C07274=1119.988,-13.062,-50.187,179.666,6.143,149.206
C07275=1119.993,-13.312,-50.175,179.666,6.138,149.205
C07276=1119.998,-13.562,-50.161,179.665,6.134,149.204
C07277=1120.003,-13.811,-50.149,179.664,6.129,149.203
C07278=1120.008,-14.061,-50.136,179.664,6.125,149.202
C07279=1120.013,-14.311,-50.123,179.663,6.120,149.202
C07280=1120.019,-14.560,-50.110,179.663,6.115,149.201
C07281=1120.023,-14.809,-50.096,179.662,6.111,149.200
C07282=1120.029,-15.058,-50.084,179.661,6.106,149.199
C07283=1120.034,-15.309,-50.070,179.661,6.101,149.198
C07284=1120.039,-15.558,-50.058,179.660,6.097,149.197
C07285=1120.044,-15.808,-50.046,179.659,6.092,149.197
C07286=1120.049,-16.058,-50.033,179.659,6.088,149.196
C07287=1120.055,-16.308,-50.020,179.658,6.082,149.195
C07288=1120.060,-16.557,-50.007,179.657,6.077,149.194
C07289=1120.065,-16.806,-49.994,179.656,6.073,149.193
C07290=1120.070,-17.056,-49.981,179.656,6.068,149.192
C07291=1120.075,-17.306,-49.968,179.655,6.064,149.192
C07292=1120.081,-17.555,-49.956,179.655,6.059,149.191
C07293=1120.085,-17.805,-49.943,179.654,6.054,149.190
C07294=1120.090,-18.054,-49.930,179.653,6.050,149.189
C07295=1120.095,-18.304,-49.918,179.653,6.045,149.188
C07296=1120.101,-18.553,-49.904,179.652,6.040,149.187
C07297=1120.106,-18.803,-49.891,179.652,6.036,149.186
C07298=1120.111,-19.053,-49.879,179.651,6.031,149.186
C07299=1120.116,-19.268,-49.868,179.650,6.026,149.185
C07300=1120.120,-19.484,-49.858,179.650,6.023,149.184
C07301=1120.124,-19.698,-49.846,179.649,6.019,149.183
C07302=1120.130,-19.913,-49.836,179.649,6.015,149.183
C07303=1120.133,-20.128,-49.825,179.648,6.010,149.182
C07304=1120.138,-20.343,-49.814,179.647,6.006,149.181
C07305=1120.143,-20.558,-49.803,179.647,6.002,149.181
C07306=1120.147,-20.774,-49.792,179.646,5.998,149.180
C07307=1120.152,-21.023,-49.780,179.645,5.993,149.179
C07308=1120.158,-21.272,-49.767,179.645,5.989,149.178
C07309=1120.163,-21.522,-49.755,179.644,5.984,149.177
C07310=1120.167,-21.772,-49.742,179.644,5.979,149.176
C07311=1120.173,-22.022,-49.729,179.643,5.974,149.175
C07312=1120.178,-22.271,-49.717,179.643,5.970,149.175
C07313=1120.183,-22.521,-49.705,179.642,5.964,149.174
C07314=1120.188,-22.770,-49.692,179.641,5.960,149.173
C07315=1120.193,-23.020,-49.680,179.640,5.955,149.172
C07316=1120.199,-23.270,-49.668,179.640,5.950,149.171
C07317=1120.203,-23.520,-49.655,179.640,5.946,149.170
C07318=1120.208,-23.769,-49.642,179.638,5.940,149.169
C07319=1120.215,-24.019,-49.630,179.638,5.935,149.168
C07320=1120.220,-24.268,-49.617,179.637,5.931,149.168
C07321=1120.225,-24.518,-49.604,179.637,5.926,149.167
C07322=1120.230,-24.768,-49.593,179.637,5.921,149.166
C07323=1120.235,-25.017,-49.580,179.635,5.916,149.165
C07324=1120.241,-25.266,-49.567,179.635,5.911,149.164
C07325=1120.245,-25.517,-49.555,179.635,5.906,149.163
C07326=1120.251,-25.766,-49.542,179.634,5.902,149.162
C07327=1120.256,-26.016,-49.531,179.634,5.897,149.161
C07328=1120.261,-26.266,-49.518,179.634,5.892,149.160
C07329=1120.266,-26.515,-49.507,179.635,5.889,149.159
C07330=1120.271,-26.764,-49.494,179.636,5.884,149.158
C07331=1120.276,-27.014,-49.481,179.636,5.880,149.157
C07332=1120.281,-27.264,-49.470,179.637,5.876,149.156
C07333=1120.287,-27.513,-49.457,179.637,5.872,149.155
C07334=1120.292,-27.763,-49.445,179.638,5.868,149.154
C07335=1120.297,-28.013,-49.432,179.638,5.864,149.153
C07336=1120.302,-28.263,-49.420,179.639,5.859,149.152
C07337=1120.307,-28.512,-49.408,179.639,5.855,149.151
C07338=1120.313,-28.762,-49.396,179.640,5.851,149.150
C07339=1120.318,-29.012,-49.383,179.640,5.847,149.149
C07340=1120.323,-29.261,-49.371,179.640,5.843,149.148
C07341=1120.328,-29.511,-49.359,179.640,5.839,149.147
C07342=1120.334,-29.761,-49.347,179.641,5.835,149.146
C07343=1120.339,-30.010,-49.334,179.641,5.831,149.145
C07344=1120.344,-30.260,-49.322,179.641,5.826,149.144
C07345=1120.349,-30.509,-49.310,179.641,5.822,149.143
C07346=1120.354,-30.759,-49.298,179.641,5.818,149.142
C07347=1120.359,-31.008,-49.286,179.641,5.813,149.141
C07348=1120.365,-31.258,-49.274,179.641,5.809,149.140
C07349=1120.370,-31.507,-49.261,179.641,5.805,149.139
C07350=1120.375,-31.757,-49.249,179.641,5.800,149.138
C07351=1120.381,-32.007,-49.238,179.641,5.796,149.137
C07352=1120.386,-32.257,-49.225,179.641,5.791,149.136
C07353=1120.390,-32.506,-49.214,179.641,5.787,149.135
C07354=1120.395,-32.756,-49.201,179.640,5.783,149.135
C07355=1120.400,-32.972,-49.190,179.640,5.779,149.134
C07356=1120.404,-33.186,-49.180,179.640,5.776,149.133
C07357=1120.409,-33.402,-49.170,179.640,5.772,149.132
C07358=1120.414,-33.616,-49.160,179.639,5.767,149.131
C07359=1120.417,-33.832,-49.149,179.638,5.764,149.131
C07360=1120.422,-34.047,-49.139,179.638,5.760,149.130
C07361=1120.427,-34.262,-49.129,179.638,5.756,149.129
C07362=1120.432,-34.477,-49.118,179.637,5.752,149.129
C07363=1120.437,-34.727,-49.107,179.637,5.747,149.128
C07364=1120.442,-34.976,-49.094,179.636,5.743,149.127
C07365=1120.447,-35.226,-49.082,179.635,5.738,149.126
C07366=1120.453,-35.476,-49.070,179.635,5.733,149.125
C07367=1120.458,-35.725,-49.058,179.634,5.729,149.124
C07368=1120.462,-35.975,-49.046,179.634,5.724,149.124
C07369=1120.468,-36.225,-49.034,179.633,5.719,149.123
C07370=1120.473,-36.474,-49.022,179.632,5.715,149.122
C07371=1120.478,-36.724,-49.010,179.632,5.710,149.121
C07372=1120.483,-36.974,-48.999,179.631,5.705,149.120
C07373=1120.489,-37.224,-48.987,179.630,5.700,149.120
C07374=1120.494,-37.474,-48.975,179.629,5.696,149.119
C07375=1120.499,-37.723,-48.962,179.628,5.691,149.118
C07376=1120.504,-37.973,-48.951,179.627,5.686,149.117
C07377=1120.509,-38.223,-48.939,179.626,5.681,149.116
C07378=1120.515,-38.472,-48.928,179.625,5.676,149.115
C07379=1120.520,-38.721,-48.916,179.624,5.671,149.115
C07380=1120.525,-38.971,-48.904,179.623,5.666,149.114
C07381=1120.530,-39.221,-48.892,179.622,5.661,149.113
C07382=1120.535,-39.470,-48.881,179.621,5.655,149.112
C07383=1120.541,-39.720,-48.869,179.620,5.651,149.112
C07384=1120.546,-39.970,-48.857,179.619,5.645,149.111
C07385=1120.551,-40.220,-48.846,179.617,5.640,149.110
C07386=1120.557,-40.469,-48.834,179.616,5.635,149.109
C07387=1120.562,-40.719,-48.822,179.615,5.630,149.109
C07388=1120.567,-40.969,-48.811,179.614,5.624,149.108
C07389=1120.572,-41.219,-48.799,179.612,5.619,149.107
C07390=1120.578,-41.468,-48.787,179.611,5.613,149.106
C07391=1120.582,-41.718,-48.776,179.610,5.608,149.105
C07392=1120.588,-41.967,-48.764,179.609,5.603,149.104
C07393=1120.593,-42.217,-48.753,179.607,5.597,149.104
C07394=1120.599,-42.467,-48.741,179.605,5.591,149.103
C07395=1120.603,-42.717,-48.730,179.604,5.586,149.102
C07396=1120.609,-42.966,-48.718,179.603,5.580,149.101
C07397=1120.614,-43.215,-48.707,179.602,5.576,149.100
C07398=1120.619,-43.465,-48.695,179.602,5.570,149.099
C07399=1120.624,-43.715,-48.684,179.603,5.565,149.098
C07400=1120.630,-43.965,-48.672,179.603,5.561,149.097
C07401=1120.635,-44.215,-48.660,179.603,5.556,149.096
C07402=1120.640,-44.464,-48.649,179.603,5.552,149.095
C07403=1120.646,-44.714,-48.637,179.603,5.547,149.094
C07404=1120.650,-44.963,-48.626,179.603,5.542,149.093
C07405=1120.655,-45.214,-48.615,179.604,5.538,149.092
C07406=1120.661,-45.463,-48.604,179.604,5.533,149.091
C07407=1120.666,-45.712,-48.593,179.604,5.528,149.089
C07408=1120.672,-45.962,-48.581,179.604,5.523,149.089
C07409=1120.676,-46.212,-48.569,179.604,5.518,149.087
C07410=1120.682,-46.461,-48.558,179.605,5.514,149.086
C07411=1120.687,-46.677,-48.549,179.605,5.510,149.085
C07412=1120.691,-46.892,-48.538,179.605,5.506,149.084
C07413=1120.695,-47.108,-48.529,179.605,5.501,149.084
C07414=1120.700,-47.323,-48.519,179.605,5.497,149.083
C07415=1120.704,-47.538,-48.510,179.605,5.493,149.082
C07416=1120.709,-47.753,-48.500,179.605,5.490,149.081
C07417=1120.714,-47.968,-48.489,179.605,5.486,149.080
C07418=1120.718,-48.184,-48.480,179.606,5.482,149.079
C07419=1120.723,-48.433,-48.468,179.606,5.476,149.078
C07420=1120.728,-48.682,-48.458,179.606,5.472,149.077
C07421=1120.734,-48.933,-48.446,179.606,5.467,149.076
C07422=1120.739,-49.182,-48.435,179.607,5.463,149.075
C07423=1120.745,-49.432,-48.424,179.607,5.458,149.073
C07424=1120.749,-49.681,-48.412,179.607,5.453,149.072
C07425=1120.754,-49.931,-48.402,179.607,5.449,149.071
C07426=1120.760,-50.181,-48.390,179.607,5.444,149.070
C07427=1120.765,-50.430,-48.379,179.608,5.439,149.069
C07428=1120.771,-50.680,-48.367,179.607,5.435,149.068
C07429=1120.776,-50.930,-48.357,179.608,5.430,149.067
C07430=1120.781,-51.179,-48.345,179.608,5.425,149.066
C07431=1120.786,-51.429,-48.334,179.608,5.420,149.065
C07432=1120.792,-51.679,-48.323,179.608,5.416,149.064
C07433=1120.797,-51.929,-48.312,179.608,5.411,149.063
C07434=1120.802,-52.178,-48.300,179.609,5.407,149.062
C07435=1120.808,-52.428,-48.290,179.609,5.402,149.061
C07436=1120.812,-52.678,-48.279,179.609,5.397,149.060
C07437=1120.818,-52.928,-48.267,179.609,5.392,149.058
C07438=1120.823,-53.177,-48.257,179.609,5.388,149.057
C07439=1120.828,-53.427,-48.245,179.610,5.383,149.056
C07440=1120.834,-53.677,-48.234,179.610,5.378,149.055
C07441=1120.839,-53.926,-48.223,179.609,5.373,149.054
C07442=1120.844,-54.176,-48.212,179.610,5.369,149.053
C07443=1120.849,-54.426,-48.201,179.610,5.364,149.052
C07444=1120.855,-54.675,-48.190,179.610,5.360,149.051
C07445=1120.859,-54.925,-48.179,179.610,5.355,149.050
C07446=1120.865,-55.175,-48.168,179.611,5.350,149.049
C07447=1120.871,-55.424,-48.156,179.611,5.346,149.048
C07448=1120.876,-55.675,-48.146,179.611,5.341,149.047
C07449=1120.881,-55.924,-48.135,179.611,5.336,149.045
C07450=1120.886,-56.174,-48.124,179.611,5.331,149.045
C07451=1120.891,-56.424,-48.112,179.612,5.327,149.043
C07452=1120.897,-56.673,-48.102,179.612,5.322,149.042
C07453=1120.902,-56.923,-48.091,179.612,5.318,149.041
C07454=1120.907,-57.173,-48.081,179.612,5.313,149.040
C07455=1120.912,-57.422,-48.069,179.612,5.308,149.039
C07456=1120.917,-57.672,-48.058,179.612,5.304,149.038
C07457=1120.923,-57.922,-48.047,179.612,5.299,149.037
C07458=1120.928,-58.172,-48.037,179.613,5.295,149.036
C07459=1120.933,-58.421,-48.026,179.613,5.289,149.035
C07460=1120.938,-58.671,-48.015,179.613,5.284,149.034
C07461=1120.944,-58.920,-48.004,179.613,5.280,149.033
C07462=1120.949,-59.171,-47.993,179.613,5.275,149.032
C07463=1120.954,-59.420,-47.982,179.614,5.271,149.031
C07464=1120.959,-59.670,-47.972,179.613,5.266,149.030
C07465=1120.964,-59.919,-47.960,179.614,5.262,149.028
C07466=1120.970,-60.169,-47.950,179.614,5.257,149.028
C07467=1120.974,-60.384,-47.941,179.613,5.252,149.027
C07468=1120.979,-60.600,-47.932,179.612,5.248,149.026
C07469=1120.983,-60.815,-47.922,179.612,5.243,149.025
C07470=1120.988,-61.030,-47.912,179.611,5.239,149.024
C07471=1120.993,-61.246,-47.903,179.610,5.234,149.024
C07472=1120.997,-61.461,-47.894,179.610,5.230,149.023
C07473=1121.001,-61.676,-47.885,179.609,5.225,149.022
C07474=1121.006,-61.892,-47.876,179.609,5.221,149.021
C07475=1121.011,-62.141,-47.865,179.608,5.216,149.020
C07476=1121.016,-62.391,-47.854,179.607,5.210,149.019
C07477=1121.022,-62.641,-47.844,179.607,5.205,149.018
C07478=1121.027,-62.890,-47.832,179.606,5.200,149.017
C07479=1121.033,-63.140,-47.822,179.606,5.195,149.017
C07480=1121.038,-63.390,-47.811,179.605,5.190,149.016
C07481=1121.043,-63.640,-47.801,179.605,5.184,149.014
C07482=1121.048,-63.889,-47.790,179.604,5.179,149.014
C07483=1121.054,-64.139,-47.780,179.603,5.174,149.013
C07484=1121.059,-64.389,-47.770,179.602,5.169,149.012
C07485=1121.064,-64.639,-47.759,179.602,5.164,149.011
C07486=1121.070,-64.888,-47.748,179.601,5.158,149.010
C07487=1121.075,-65.138,-47.737,179.601,5.153,149.009
C07488=1121.080,-65.387,-47.727,179.600,5.147,149.008
C07489=1121.085,-65.638,-47.717,179.600,5.142,149.007
C07490=1121.090,-65.887,-47.706,179.599,5.137,149.006
C07491=1121.096,-66.136,-47.696,179.599,5.132,149.005
C07492=1121.101,-66.386,-47.685,179.598,5.126,149.004
C07493=1121.107,-66.636,-47.675,179.598,5.121,149.003
C07494=1121.112,-66.886,-47.664,179.598,5.117,149.002
C07495=1121.117,-67.136,-47.654,179.597,5.111,149.001
C07496=1121.123,-67.385,-47.644,179.597,5.106,149.000
C07497=1121.128,-67.635,-47.632,179.596,5.100,148.999
C07498=1121.133,-67.884,-47.622,179.596,5.095,148.998
C07499=1121.138,-68.135,-47.612,179.596,5.089,148.997
C07500=1121.143,-68.384,-47.602,179.595,5.084,148.996
C07501=1121.149,-68.634,-47.592,179.595,5.080,148.995
C07502=1121.154,-68.884,-47.581,179.594,5.074,148.994
C07503=1121.159,-69.133,-47.571,179.594,5.069,148.992
C07504=1121.165,-69.383,-47.561,179.594,5.064,148.991
C07505=1121.170,-69.633,-47.550,179.594,5.058,148.990
C07506=1121.175,-69.883,-47.540,179.593,5.053,148.989
C07507=1121.181,-70.132,-47.530,179.593,5.047,148.988
C07508=1121.186,-70.382,-47.519,179.592,5.042,148.987
C07509=1121.191,-70.632,-47.510,179.593,5.037,148.986
C07510=1121.196,-70.881,-47.499,179.592,5.031,148.985
C07511=1121.201,-71.131,-47.489,179.592,5.026,148.984
C07512=1121.207,-71.381,-47.479,179.592,5.021,148.983
C07513=1121.213,-71.631,-47.468,179.591,5.017,148.982
C07514=1121.218,-71.881,-47.458,179.591,5.011,148.981
C07515=1121.223,-72.130,-47.448,179.591,5.005,148.980
C07516=1121.228,-72.380,-47.438,179.591,5.000,148.978
C07517=1121.233,-72.630,-47.428,179.590,4.995,148.978
C07518=1121.239,-72.879,-47.417,179.590,4.990,148.976
C07519=1121.245,-73.130,-47.408,179.591,4.984,148.975
C07520=1121.250,-73.379,-47.398,179.590,4.980,148.974
C07521=1121.254,-73.629,-47.388,179.590,4.974,148.973
C07522=1121.260,-73.879,-47.377,179.590,4.968,148.972
C07523=1121.265,-74.094,-47.368,179.590,4.965,148.971
C07524=1121.269,-74.309,-47.361,179.590,4.960,148.970
C07525=1121.274,-74.525,-47.351,179.589,4.955,148.969
C07526=1121.278,-74.740,-47.343,179.590,4.951,148.968
C07527=1121.283,-74.956,-47.334,179.590,4.946,148.967
C07528=1121.287,-75.170,-47.326,179.590,4.942,148.966
C07529=1121.292,-75.386,-47.317,179.590,4.937,148.965
C07530=1121.297,-75.602,-47.308,179.589,4.932,148.964
C07531=1121.302,-75.851,-47.298,179.590,4.927,148.963
C07532=1121.308,-76.101,-47.288,179.590,4.922,148.962
C07533=1121.313,-76.351,-47.278,179.590,4.917,148.961
C07534=1121.318,-76.601,-47.268,179.590,4.912,148.960
C07535=1121.323,-76.850,-47.258,179.590,4.907,148.958
C07536=1121.329,-77.100,-47.248,179.590,4.902,148.958
C07537=1121.335,-77.350,-47.239,179.589,4.896,148.956
C07538=1121.340,-77.599,-47.229,179.590,4.891,148.955
C07539=1121.345,-77.850,-47.218,179.590,4.886,148.954
C07540=1121.350,-78.099,-47.208,179.590,4.880,148.953
C07541=1121.355,-78.349,-47.199,179.590,4.875,148.952
C07542=1121.361,-78.599,-47.189,179.590,4.870,148.951
C07543=1121.367,-78.848,-47.179,179.590,4.865,148.949
C07544=1121.372,-79.098,-47.170,179.590,4.860,148.948
C07545=1121.377,-79.348,-47.159,179.591,4.855,148.947
C07546=1121.382,-79.597,-47.150,179.591,4.849,148.946
C07547=1121.388,-79.848,-47.140,179.591,4.844,148.945
C07548=1121.393,-80.097,-47.130,179.591,4.839,148.944
C07549=1121.398,-80.346,-47.120,179.591,4.834,148.942
C07550=1121.404,-80.596,-47.111,179.591,4.829,148.941
C07551=1121.410,-80.846,-47.101,179.592,4.824,148.940
C07552=1121.414,-81.097,-47.091,179.592,4.819,148.939
C07553=1121.420,-81.346,-47.081,179.592,4.813,148.938
C07554=1121.425,-81.595,-47.072,179.592,4.808,148.936
C07555=1121.430,-81.846,-47.062,179.592,4.803,148.935
C07556=1121.435,-82.095,-47.053,179.592,4.798,148.934
C07557=1121.441,-82.345,-47.043,179.593,4.793,148.933
C07558=1121.447,-82.594,-47.033,179.593,4.788,148.932
C07559=1121.451,-82.844,-47.023,179.594,4.783,148.930
C07560=1121.457,-83.095,-47.013,179.594,4.778,148.929
C07561=1121.462,-83.344,-47.004,179.594,4.773,148.928
C07562=1121.468,-83.594,-46.994,179.595,4.767,148.927
C07563=1121.473,-83.843,-46.985,179.595,4.762,148.926
C07564=1121.479,-84.093,-46.975,179.595,4.757,148.925
C07565=1121.483,-84.343,-46.966,179.596,4.753,148.923
C07566=1121.489,-84.593,-46.956,179.596,4.748,148.922
C07567=1121.494,-84.842,-46.946,179.596,4.742,148.921
C07568=1121.500,-85.092,-46.937,179.597,4.737,148.920
C07569=1121.505,-85.341,-46.927,179.597,4.732,148.918
C07570=1121.510,-85.592,-46.917,179.598,4.727,148.917
C07571=1121.515,-85.841,-46.908,179.598,4.722,148.916
C07572=1121.521,-86.092,-46.898,179.598,4.717,148.915
C07573=1121.526,-86.341,-46.889,179.598,4.712,148.914
C07574=1121.532,-86.591,-46.879,179.599,4.707,148.912
C07575=1121.537,-86.840,-46.870,179.600,4.702,148.911
C07576=1121.543,-87.090,-46.860,179.600,4.697,148.910
C07577=1121.548,-87.340,-46.851,179.601,4.692,148.909
C07578=1121.553,-87.589,-46.842,179.601,4.687,148.908
C07579=1121.557,-87.806,-46.833,179.602,4.683,148.906
C07580=1121.562,-88.021,-46.825,179.602,4.679,148.905
C07581=1121.567,-88.236,-46.817,179.603,4.675,148.904
C07582=1121.572,-88.451,-46.809,179.602,4.670,148.903
C07583=1121.576,-88.667,-46.801,179.603,4.665,148.902
C07584=1121.580,-88.883,-46.793,179.603,4.662,148.901
C07585=1121.585,-89.098,-46.785,179.604,4.657,148.900
C07586=1121.590,-89.314,-46.776,179.604,4.653,148.899
C07587=1121.595,-89.563,-46.767,179.605,4.648,148.898
C07588=1121.601,-89.813,-46.757,179.605,4.644,148.897
C07589=1121.606,-90.063,-46.748,179.606,4.638,148.895
C07590=1121.611,-90.313,-46.739,179.607,4.634,148.894
C07591=1121.617,-90.563,-46.729,179.607,4.629,148.893
C07592=1121.622,-90.813,-46.720,179.608,4.624,148.892
C07593=1121.627,-91.062,-46.711,179.608,4.619,148.890
C07594=1121.633,-91.312,-46.701,179.609,4.614,148.889
C07595=1121.638,-91.562,-46.692,179.609,4.609,148.888
C07596=1121.643,-91.811,-46.682,179.610,4.605,148.887
C07597=1121.649,-92.061,-46.673,179.610,4.600,148.886
C07598=1121.654,-92.311,-46.664,179.612,4.595,148.884
C07599=1121.659,-92.561,-46.654,179.612,4.590,148.883
C07600=1121.664,-92.810,-46.645,179.613,4.585,148.882
C07601=1121.670,-93.060,-46.636,179.613,4.581,148.881
C07602=1121.676,-93.310,-46.627,179.614,4.576,148.879
C07603=1121.680,-93.560,-46.617,179.615,4.571,148.878
C07604=1121.686,-93.810,-46.608,179.615,4.566,148.877
C07605=1121.691,-94.060,-46.599,179.616,4.562,148.876
C07606=1121.697,-94.310,-46.590,179.617,4.557,148.874
C07607=1121.701,-94.559,-46.580,179.617,4.552,148.873
C07608=1121.708,-94.808,-46.571,179.618,4.548,148.872
C07609=1121.713,-95.058,-46.562,179.618,4.543,148.871
C07610=1121.718,-95.308,-46.553,179.618,4.537,148.870
C07611=1121.723,-95.557,-46.544,179.618,4.532,148.869
C07612=1121.729,-95.807,-46.534,179.619,4.528,148.867
C07613=1121.734,-96.057,-46.525,179.619,4.523,148.866
C07614=1121.739,-96.307,-46.517,179.620,4.518,148.865
C07615=1121.745,-96.557,-46.507,179.620,4.512,148.864
C07616=1121.750,-96.807,-46.498,179.620,4.507,148.863
C07617=1121.755,-97.056,-46.489,179.621,4.503,148.861
C07618=1121.761,-97.306,-46.480,179.621,4.498,148.860
C07619=1121.766,-97.556,-46.470,179.621,4.493,148.859
C07620=1121.772,-97.806,-46.461,179.621,4.487,148.858
C07621=1121.777,-98.055,-46.453,179.622,4.483,148.857
C07622=1121.783,-98.305,-46.444,179.622,4.478,148.856
C07623=1121.788,-98.555,-46.434,179.622,4.473,148.855
C07624=1121.794,-98.805,-46.425,179.622,4.468,148.853
C07625=1121.798,-99.054,-46.416,179.623,4.463,148.852
C07626=1121.804,-99.304,-46.407,179.623,4.458,148.851
C07627=1121.810,-99.554,-46.397,179.624,4.453,148.850
C07628=1121.815,-99.804,-46.389,179.624,4.448,148.849
C07629=1121.820,-100.053,-46.380,179.624,4.443,148.847
C07630=1121.826,-100.303,-46.371,179.624,4.438,148.846
C07631=1121.831,-100.553,-46.362,179.625,4.433,148.845
C07632=1121.837,-100.803,-46.353,179.625,4.428,148.844
C07633=1121.842,-101.053,-46.344,179.625,4.423,148.843
C07634=1121.847,-101.303,-46.335,179.625,4.418,148.842
C07635=1121.852,-101.518,-46.327,179.626,4.414,148.840
C07636=1121.856,-101.734,-46.319,179.626,4.409,148.840
C07637=1121.861,-101.949,-46.312,179.626,4.405,148.839
C07638=1121.865,-102.165,-46.304,179.626,4.401,148.838
C07639=1121.870,-102.381,-46.297,179.627,4.396,148.836
C07640=1121.874,-102.596,-46.289,179.627,4.392,148.835
C07641=1121.879,-102.811,-46.281,179.627,4.388,148.835
C07642=1121.883,-103.027,-46.273,179.627,4.383,148.834
C07643=1121.889,-103.276,-46.265,179.627,4.378,148.832
C07644=1121.895,-103.527,-46.255,179.628,4.374,148.831
C07645=1121.900,-103.776,-46.246,179.628,4.369,148.830
C07646=1121.906,-104.027,-46.238,179.628,4.363,148.829
C07647=1121.911,-104.277,-46.229,179.629,4.358,148.828
C07648=1121.917,-104.526,-46.221,179.629,4.353,148.826
C07649=1121.922,-104.776,-46.212,179.629,4.348,148.825
C07650=1121.927,-105.026,-46.203,179.629,4.343,148.824
C07651=1121.932,-105.275,-46.194,179.630,4.338,148.823
C07652=1121.937,-105.525,-46.185,179.630,4.332,148.822
C07653=1121.943,-105.774,-46.177,179.630,4.327,148.820
C07654=1121.948,-106.024,-46.168,179.631,4.323,148.819
C07655=1121.953,-106.274,-46.159,179.631,4.318,148.818
C07656=1121.959,-106.525,-46.151,179.631,4.313,148.817
C07657=1121.964,-106.774,-46.142,179.631,4.308,148.816
C07658=1121.971,-107.024,-46.133,179.631,4.303,148.815
C07659=1121.976,-107.274,-46.124,179.632,4.297,148.814
C07660=1121.981,-107.524,-46.115,179.632,4.292,148.812
C07661=1121.986,-107.773,-46.106,179.632,4.287,148.811
C07662=1121.992,-108.023,-46.098,179.632,4.282,148.810
C07663=1121.997,-108.273,-46.089,179.633,4.277,148.809
C07664=1122.002,-108.523,-46.080,179.633,4.272,148.808
C07665=1122.008,-108.773,-46.071,179.633,4.266,148.806
C07666=1122.013,-109.022,-46.063,179.633,4.261,148.805
C07667=1122.019,-109.272,-46.055,179.634,4.256,148.804
C07668=1122.024,-109.522,-46.046,179.634,4.251,148.803
C07669=1122.030,-109.771,-46.037,179.634,4.246,148.802
C07670=1122.034,-110.021,-46.029,179.634,4.241,148.800
C07671=1122.040,-110.271,-46.021,179.635,4.235,148.799
C07672=1122.045,-110.521,-46.012,179.635,4.230,148.798
C07673=1122.051,-110.770,-46.003,179.635,4.225,148.797
C07674=1122.056,-111.020,-45.994,179.635,4.220,148.796
C07675=1122.061,-111.271,-45.986,179.636,4.215,148.794
C07676=1122.067,-111.520,-45.978,179.636,4.210,148.793
C07677=1122.072,-111.770,-45.969,179.636,4.204,148.792
C07678=1122.078,-112.020,-45.961,179.636,4.199,148.791
C07679=1122.083,-112.269,-45.952,179.636,4.194,148.790
C07680=1122.089,-112.519,-45.943,179.636,4.189,148.789
C07681=1122.094,-112.770,-45.935,179.637,4.184,148.787
C07682=1122.100,-113.019,-45.926,179.637,4.179,148.786
C07683=1122.105,-113.269,-45.918,179.637,4.174,148.785
C07684=1122.110,-113.519,-45.910,179.637,4.169,148.784
C07685=1122.116,-113.768,-45.901,179.638,4.163,148.783
C07686=1122.121,-114.018,-45.893,179.638,4.158,148.781
C07687=1122.126,-114.268,-45.884,179.638,4.152,148.780
C07688=1122.132,-114.517,-45.876,179.638,4.147,148.779
C07689=1122.137,-114.768,-45.868,179.638,4.142,148.778
C07690=1122.143,-115.017,-45.859,179.638,4.137,148.777
C07691=1122.147,-115.233,-45.852,179.639,4.132,148.775
C07692=1122.152,-115.448,-45.845,179.639,4.128,148.774
C07693=1122.157,-115.664,-45.838,179.639,4.124,148.773
C07694=1122.161,-115.880,-45.830,179.640,4.118,148.772
C07695=1122.166,-116.096,-45.823,179.639,4.114,148.771
C07696=1122.171,-116.311,-45.816,179.640,4.109,148.770
C07697=1122.175,-116.527,-45.809,179.640,4.104,148.769
C07698=1122.180,-116.742,-45.802,179.640,4.101,148.768
C07699=1122.185,-116.992,-45.793,179.641,4.095,148.767
C07700=1122.191,-117.242,-45.785,179.641,4.090,148.766
C07701=1122.196,-117.492,-45.776,179.641,4.084,148.765
C07702=1122.202,-117.741,-45.769,179.641,4.079,148.763
C07703=1122.207,-117.991,-45.760,179.641,4.074,148.762
C07704=1122.213,-118.241,-45.752,179.641,4.069,148.761
C07705=1122.218,-118.491,-45.744,179.642,4.063,148.759
C07706=1122.223,-118.741,-45.736,179.642,4.058,148.758
C07707=1122.229,-118.991,-45.728,179.642,4.052,148.757
C07708=1122.234,-119.241,-45.719,179.642,4.047,148.756
C07709=1122.240,-119.490,-45.711,179.643,4.042,148.755
C07710=1122.245,-119.740,-45.703,179.643,4.036,148.753
C07711=1122.251,-119.990,-45.695,179.643,4.031,148.752
C07712=1122.256,-120.240,-45.687,179.643,4.025,148.751
C07713=1122.262,-120.489,-45.678,179.643,4.020,148.750
C07714=1122.267,-120.739,-45.671,179.643,4.015,148.749
C07715=1122.272,-120.989,-45.662,179.644,4.010,148.747
C07716=1122.278,-121.239,-45.654,179.643,4.004,148.746
C07717=1122.283,-121.489,-45.647,179.644,3.998,148.745
C07718=1122.288,-121.738,-45.638,179.645,3.993,148.744
C07719=1122.294,-121.989,-45.630,179.645,3.988,148.742
C07720=1122.299,-122.238,-45.623,179.645,3.982,148.741
C07721=1122.304,-122.488,-45.614,179.645,3.977,148.740
C07722=1122.310,-122.738,-45.606,179.645,3.971,148.739
C07723=1122.315,-122.988,-45.598,179.645,3.966,148.737
C07724=1122.321,-123.237,-45.590,179.646,3.960,148.736
C07725=1122.326,-123.488,-45.582,179.646,3.955,148.735
C07726=1122.332,-123.737,-45.574,179.646,3.950,148.734
C07727=1122.338,-123.987,-45.567,179.647,3.944,148.732
C07728=1122.343,-124.237,-45.558,179.646,3.938,148.731
C07729=1122.348,-124.486,-45.551,179.647,3.933,148.730
C07730=1122.354,-124.737,-45.542,179.647,3.928,148.729
C07731=1122.359,-124.986,-45.535,179.647,3.922,148.727
C07732=1122.364,-125.236,-45.526,179.647,3.916,148.726
C07733=1122.370,-125.486,-45.518,179.648,3.911,148.725
C07734=1122.375,-125.736,-45.511,179.647,3.905,148.724
C07735=1122.381,-125.986,-45.503,179.648,3.900,148.722
C07736=1122.386,-126.235,-45.495,179.649,3.895,148.721
C07737=1122.392,-126.485,-45.487,179.648,3.889,148.720
C07738=1122.397,-126.735,-45.480,179.649,3.883,148.719
C07739=1122.402,-126.985,-45.471,179.648,3.877,148.717
C07740=1122.408,-127.234,-45.464,179.649,3.872,148.716
C07741=1122.413,-127.485,-45.456,179.649,3.867,148.715
C07742=1122.419,-127.734,-45.448,179.649,3.861,148.713
C07743=1122.424,-127.984,-45.440,179.649,3.855,148.712
C07744=1122.430,-128.234,-45.432,179.649,3.849,148.711
C07745=1122.435,-128.483,-45.425,179.650,3.844,148.710
C07746=1122.441,-128.734,-45.417,179.650,3.839,148.708
C07747=1122.017,-128.724,-45.443,179.657,3.843,148.707
C07748=1122.013,-128.474,-45.451,179.657,3.849,148.708
C07749=1122.006,-128.224,-45.459,179.657,3.854,148.710
C07750=1122.001,-127.975,-45.466,179.657,3.860,148.711
C07751=1121.996,-127.725,-45.474,179.656,3.865,148.712
C07752=1121.990,-127.475,-45.482,179.656,3.870,148.713
C07753=1121.985,-127.225,-45.490,179.656,3.876,148.715
C07754=1121.980,-126.975,-45.497,179.656,3.882,148.716
C07755=1121.974,-126.725,-45.506,179.655,3.887,148.717
C07756=1121.968,-126.476,-45.514,179.656,3.893,148.719
C07757=1121.963,-126.226,-45.521,179.655,3.898,148.720
C07758=1121.957,-125.976,-45.529,179.655,3.904,148.721
C07759=1121.952,-125.727,-45.537,179.655,3.910,148.722
C07760=1121.947,-125.476,-45.545,179.654,3.915,148.724
C07761=1121.942,-125.227,-45.553,179.655,3.921,148.725
C07762=1121.936,-124.976,-45.561,179.654,3.926,148.726
C07763=1121.930,-124.727,-45.569,179.654,3.931,148.727
C07764=1121.926,-124.477,-45.577,179.654,3.937,148.728
C07765=1121.920,-124.227,-45.585,179.654,3.943,148.730
C07766=1121.914,-123.977,-45.593,179.653,3.948,148.731
C07767=1121.909,-123.728,-45.601,179.653,3.953,148.732
C07768=1121.904,-123.477,-45.609,179.653,3.959,148.734
C07769=1121.898,-123.228,-45.617,179.653,3.965,148.735
C07770=1121.893,-122.978,-45.625,179.653,3.970,148.736
C07771=1121.887,-122.728,-45.633,179.652,3.975,148.737
C07772=1121.882,-122.478,-45.641,179.652,3.981,148.739
C07773=1121.877,-122.229,-45.649,179.652,3.986,148.740
C07774=1121.871,-121.979,-45.657,179.652,3.992,148.741
C07775=1121.865,-121.729,-45.665,179.651,3.997,148.742
C07776=1121.861,-121.479,-45.673,179.652,4.003,148.743
C07777=1121.854,-121.230,-45.681,179.651,4.008,148.745
C07778=1121.849,-120.980,-45.690,179.651,4.013,148.746
C07779=1121.844,-120.730,-45.697,179.650,4.019,148.747
C07780=1121.839,-120.480,-45.705,179.650,4.025,148.749
C07781=1121.833,-120.231,-45.714,179.650,4.030,148.750
C07782=1121.827,-119.980,-45.722,179.650,4.035,148.751
C07783=1121.822,-119.731,-45.730,179.650,4.040,148.752
C07784=1121.817,-119.481,-45.738,179.649,4.045,148.753
C07785=1121.812,-119.231,-45.747,179.650,4.051,148.755
C07786=1121.806,-118.981,-45.755,179.649,4.057,148.756
C07787=1121.801,-118.732,-45.763,179.649,4.062,148.757
C07788=1121.795,-118.482,-45.771,179.649,4.067,148.758
C07789=1121.790,-118.232,-45.780,179.649,4.072,148.759
C07790=1121.784,-117.982,-45.788,179.648,4.077,148.761
C07791=1121.779,-117.732,-45.797,179.648,4.084,148.762
C07792=1121.774,-117.482,-45.804,179.648,4.089,148.763
C07793=1121.768,-117.233,-45.813,179.647,4.094,148.764
C07794=1121.763,-116.983,-45.821,179.647,4.099,148.766
C07795=1121.757,-116.734,-45.830,179.647,4.104,148.767
C07796=1121.752,-116.517,-45.837,179.647,4.109,148.768
C07797=1121.748,-116.302,-45.843,179.647,4.113,148.769
C07798=1121.743,-116.087,-45.851,179.647,4.118,148.770
C07799=1121.739,-115.870,-45.858,179.646,4.122,148.771
C07800=1121.734,-115.655,-45.866,179.646,4.127,148.772
C07801=1121.729,-115.439,-45.872,179.646,4.131,148.773
C07802=1121.724,-115.224,-45.880,179.646,4.136,148.774
C07803=1121.720,-115.008,-45.887,179.646,4.140,148.775
C07804=1121.715,-114.758,-45.896,179.646,4.146,148.776
C07805=1121.709,-114.509,-45.903,179.646,4.151,148.777
C07806=1121.704,-114.259,-45.912,179.645,4.157,148.779
C07807=1121.699,-114.009,-45.921,179.645,4.162,148.780
C07808=1121.692,-113.759,-45.929,179.644,4.167,148.781
C07809=1121.687,-113.509,-45.938,179.644,4.172,148.783
C07810=1121.682,-113.259,-45.947,179.644,4.178,148.784
C07811=1121.676,-113.010,-45.955,179.644,4.183,148.785
C07812=1121.671,-112.760,-45.964,179.643,4.188,148.786
C07813=1121.666,-112.510,-45.972,179.643,4.193,148.787
C07814=1121.660,-112.260,-45.980,179.643,4.198,148.789
C07815=1121.655,-112.011,-45.989,179.643,4.203,148.789
C07816=1121.650,-111.761,-45.998,179.643,4.208,148.791
C07817=1121.644,-111.511,-46.005,179.642,4.213,148.792
C07818=1121.639,-111.261,-46.014,179.642,4.219,148.793
C07819=1121.634,-111.011,-46.023,179.642,4.224,148.794
C07820=1121.628,-110.762,-46.032,179.642,4.229,148.795
C07821=1121.622,-110.512,-46.040,179.641,4.234,148.797
C07822=1121.617,-110.262,-46.049,179.641,4.239,148.798
C07823=1121.612,-110.012,-46.058,179.641,4.244,148.799
C07824=1121.606,-109.763,-46.066,179.641,4.250,148.800
C07825=1121.601,-109.512,-46.074,179.640,4.255,148.801
C07826=1121.596,-109.262,-46.083,179.640,4.260,148.803
C07827=1121.591,-109.013,-46.092,179.640,4.265,148.804
C07828=1121.585,-108.763,-46.101,179.640,4.270,148.805
C07829=1121.580,-108.514,-46.110,179.639,4.275,148.806
C07830=1121.574,-108.263,-46.118,179.639,4.281,148.807
C07831=1121.569,-108.013,-46.127,179.639,4.286,148.809
C07832=1121.563,-107.764,-46.135,179.639,4.291,148.810
C07833=1121.558,-107.514,-46.144,179.639,4.296,148.811
C07834=1121.553,-107.264,-46.153,179.638,4.301,148.812
C07835=1121.548,-107.015,-46.162,179.638,4.306,148.813
C07836=1121.542,-106.765,-46.170,179.638,4.312,148.815
C07837=1121.536,-106.515,-46.179,179.638,4.317,148.816
C07838=1121.531,-106.265,-46.187,179.637,4.322,148.817
C07839=1121.526,-106.015,-46.196,179.637,4.327,148.818
C07840=1121.521,-105.765,-46.205,179.637,4.332,148.819
C07841=1121.514,-105.516,-46.214,179.637,4.336,148.820
C07842=1121.509,-105.266,-46.223,179.636,4.341,148.822
C07843=1121.504,-105.016,-46.232,179.636,4.347,148.823
C07844=1121.499,-104.766,-46.241,179.636,4.352,148.824
C07845=1121.494,-104.517,-46.250,179.636,4.357,148.825
C07846=1121.488,-104.267,-46.259,179.635,4.362,148.826
C07847=1121.483,-104.018,-46.267,179.635,4.367,148.828
C07848=1121.478,-103.768,-46.276,179.635,4.372,148.829
C07849=1121.472,-103.518,-46.285,179.635,4.378,148.830
C07850=1121.467,-103.268,-46.294,179.634,4.382,148.831
C07851=1121.461,-103.018,-46.304,179.634,4.387,148.832
C07852=1121.456,-102.802,-46.311,179.634,4.392,148.833
C07853=1121.451,-102.587,-46.318,179.634,4.396,148.834
C07854=1121.447,-102.371,-46.326,179.633,4.400,148.835
C07855=1121.442,-102.156,-46.334,179.633,4.405,148.836
C07856=1121.438,-101.940,-46.342,179.633,4.409,148.837
C07857=1121.433,-101.725,-46.349,179.632,4.413,148.838
C07858=1121.429,-101.509,-46.357,179.632,4.418,148.839
C07859=1121.424,-101.294,-46.364,179.632,4.422,148.840
C07860=1121.419,-101.044,-46.374,179.632,4.427,148.842
C07861=1121.414,-100.795,-46.383,179.631,4.432,148.843
C07862=1121.408,-100.544,-46.392,179.631,4.437,148.844
C07863=1121.403,-100.295,-46.401,179.631,4.442,148.845
C07864=1121.398,-100.045,-46.410,179.631,4.447,148.846
C07865=1121.393,-99.795,-46.419,179.631,4.452,148.847
C07866=1121.386,-99.545,-46.428,179.630,4.457,148.849
C07867=1121.381,-99.296,-46.437,179.630,4.462,148.850
C07868=1121.376,-99.046,-46.446,179.629,4.467,148.851
C07869=1121.371,-98.796,-46.455,179.629,4.472,148.852
C07870=1121.365,-98.546,-46.464,179.629,4.477,148.853
C07871=1121.360,-98.296,-46.474,179.629,4.482,148.854
C07872=1121.355,-98.047,-46.483,179.628,4.487,148.856
C07873=1121.350,-97.797,-46.492,179.628,4.492,148.857
C07874=1121.344,-97.547,-46.501,179.627,4.497,148.858
C07875=1121.338,-97.297,-46.510,179.627,4.502,148.859
C07876=1121.333,-97.048,-46.519,179.627,4.507,148.860
C07877=1121.328,-96.798,-46.528,179.627,4.511,148.861
C07878=1121.322,-96.548,-46.538,179.626,4.516,148.863
C07879=1121.317,-96.298,-46.547,179.626,4.521,148.864
C07880=1121.312,-96.049,-46.555,179.626,4.527,148.865
C07881=1121.306,-95.798,-46.565,179.625,4.531,148.866
C07882=1121.301,-95.549,-46.575,179.625,4.536,148.867
C07883=1121.296,-95.299,-46.583,179.625,4.541,148.868
C07884=1121.290,-95.049,-46.593,179.625,4.546,148.870
C07885=1121.285,-94.799,-46.602,179.624,4.551,148.871
C07886=1121.280,-94.550,-46.611,179.624,4.556,148.872
C07887=1121.275,-94.300,-46.620,179.623,4.561,148.873
C07888=1121.269,-94.050,-46.630,179.623,4.565,148.874
C07889=1121.264,-93.800,-46.639,179.622,4.570,148.876
C07890=1121.258,-93.551,-46.649,179.622,4.575,148.877
C07891=1121.253,-93.301,-46.658,179.620,4.580,148.878
C07892=1121.248,-93.051,-46.667,179.620,4.585,148.879
C07893=1121.242,-92.801,-46.677,179.619,4.589,148.881
C07894=1121.237,-92.552,-46.686,179.619,4.594,148.882
C07895=1121.232,-92.302,-46.695,179.618,4.599,148.883
C07896=1121.226,-92.051,-46.704,179.617,4.603,148.884
C07897=1121.221,-91.802,-46.714,179.617,4.609,148.886
C07898=1121.216,-91.552,-46.723,179.616,4.613,148.887
C07899=1121.210,-91.302,-46.732,179.616,4.618,148.888
C07900=1121.205,-91.053,-46.742,179.615,4.623,148.889
C07901=1121.199,-90.803,-46.751,179.614,4.628,148.891
C07902=1121.194,-90.553,-46.760,179.614,4.632,148.892
C07903=1121.189,-90.304,-46.770,179.613,4.638,148.893
C07904=1121.183,-90.054,-46.779,179.613,4.642,148.894
C07905=1121.178,-89.804,-46.789,179.612,4.647,148.895
C07906=1121.172,-89.554,-46.798,179.611,4.652,148.897
C07907=1121.167,-89.304,-46.807,179.611,4.657,148.898
C07908=1121.163,-89.090,-46.816,179.610,4.661,148.899
C07909=1121.158,-88.874,-46.824,179.610,4.665,148.900
C07910=1121.154,-88.658,-46.832,179.609,4.670,148.901
C07911=1121.149,-88.443,-46.840,179.609,4.674,148.902
C07912=1121.144,-88.227,-46.849,179.609,4.678,148.903
C07913=1121.139,-88.012,-46.857,179.608,4.683,148.904
C07914=1121.135,-87.796,-46.865,179.608,4.687,148.905
C07915=1121.131,-87.581,-46.873,179.607,4.691,148.906
C07916=1121.125,-87.331,-46.883,179.607,4.696,148.908
C07917=1121.120,-87.081,-46.892,179.606,4.701,148.909
C07918=1121.114,-86.832,-46.902,179.606,4.706,148.910
C07919=1121.109,-86.582,-46.911,179.606,4.711,148.911
C07920=1121.104,-86.332,-46.921,179.605,4.716,148.912
C07921=1121.099,-86.083,-46.930,179.605,4.721,148.914
C07922=1121.093,-85.833,-46.940,179.604,4.726,148.915
C07923=1121.088,-85.583,-46.949,179.604,4.731,148.916
C07924=1121.082,-85.334,-46.959,179.604,4.736,148.917
C07925=1121.077,-85.084,-46.968,179.603,4.741,148.919
C07926=1121.072,-84.833,-46.979,179.603,4.746,148.920
C07927=1121.067,-84.584,-46.988,179.602,4.751,148.921
C07928=1121.061,-84.334,-46.998,179.602,4.756,148.922
C07929=1121.056,-84.084,-47.007,179.602,4.762,148.923
C07930=1121.050,-83.835,-47.017,179.601,4.766,148.924
C07931=1121.045,-83.585,-47.026,179.601,4.771,148.926
C07932=1121.040,-83.335,-47.036,179.601,4.776,148.927
C07933=1121.034,-83.085,-47.046,179.601,4.781,148.928
C07934=1121.029,-82.836,-47.055,179.600,4.787,148.929
C07935=1121.024,-82.586,-47.066,179.600,4.792,148.931
C07936=1121.019,-82.336,-47.075,179.600,4.797,148.932
C07937=1121.013,-82.086,-47.085,179.599,4.802,148.933
C07938=1121.008,-81.836,-47.094,179.599,4.807,148.934
C07939=1121.002,-81.587,-47.104,179.599,4.812,148.935
C07940=1120.997,-81.337,-47.114,179.599,4.817,148.936
C07941=1120.992,-81.087,-47.123,179.598,4.822,148.938
C07942=1120.987,-80.837,-47.134,179.598,4.827,148.939
C07943=1120.982,-80.588,-47.143,179.598,4.833,148.940
C07944=1120.976,-80.338,-47.153,179.598,4.838,148.941
C07945=1120.970,-80.088,-47.163,179.598,4.843,148.942
C07946=1120.965,-79.839,-47.173,179.598,4.848,148.943
C07947=1120.960,-79.589,-47.182,179.597,4.853,148.945
C07948=1120.955,-79.339,-47.193,179.597,4.858,148.946
C07949=1120.950,-79.089,-47.202,179.597,4.863,148.947
C07950=1120.944,-78.839,-47.212,179.597,4.869,148.948
C07951=1120.938,-78.590,-47.222,179.597,4.874,148.949
C07952=1120.933,-78.340,-47.232,179.597,4.879,148.950
C07953=1120.927,-78.090,-47.241,179.596,4.884,148.952
C07954=1120.922,-77.840,-47.252,179.596,4.889,148.953
C07955=1120.918,-77.591,-47.261,179.596,4.894,148.954
C07956=1120.912,-77.341,-47.272,179.597,4.900,148.955
C07957=1120.906,-77.091,-47.281,179.596,4.906,148.956
C07958=1120.901,-76.842,-47.291,179.596,4.911,148.957
C07959=1120.896,-76.592,-47.301,179.596,4.916,148.959
C07960=1120.891,-76.342,-47.311,179.596,4.921,148.960
C07961=1120.885,-76.093,-47.322,179.596,4.926,148.961
C07962=1120.880,-75.843,-47.331,179.596,4.931,148.962
C07963=1120.875,-75.592,-47.341,179.596,4.936,148.963
C07964=1120.870,-75.378,-47.350,179.596,4.941,148.964
C07965=1120.866,-75.163,-47.359,179.597,4.946,148.965
C07966=1120.861,-74.946,-47.367,179.596,4.950,148.966
C07967=1120.856,-74.732,-47.376,179.596,4.955,148.967
C07968=1120.851,-74.516,-47.384,179.596,4.959,148.968
C07969=1120.847,-74.301,-47.393,179.596,4.963,148.969
C07970=1120.843,-74.085,-47.402,179.597,4.968,148.970
C07971=1120.837,-73.870,-47.411,179.597,4.972,148.971
C07972=1120.833,-73.620,-47.420,179.596,4.977,148.972
C07973=1120.827,-73.370,-47.431,179.597,4.983,148.973
C07974=1120.822,-73.121,-47.441,179.597,4.988,148.974
C07975=1120.817,-72.870,-47.451,179.597,4.993,148.975
C07976=1120.811,-72.621,-47.462,179.597,4.998,148.976
C07977=1120.806,-72.372,-47.471,179.597,5.004,148.977
C07978=1120.801,-72.122,-47.481,179.598,5.009,148.978
C07979=1120.796,-71.872,-47.492,179.598,5.014,148.980
C07980=1120.790,-71.622,-47.502,179.598,5.020,148.981
C07981=1120.784,-71.373,-47.512,179.598,5.025,148.982
C07982=1120.779,-71.123,-47.523,179.598,5.030,148.983
C07983=1120.774,-70.873,-47.533,179.598,5.035,148.984
C07984=1120.769,-70.624,-47.543,179.599,5.041,148.985
C07985=1120.764,-70.374,-47.553,179.599,5.046,148.986
C07986=1120.758,-70.124,-47.564,179.599,5.051,148.987
C07987=1120.753,-69.874,-47.574,179.600,5.057,148.988
C07988=1120.748,-69.624,-47.584,179.600,5.062,148.989
C07989=1120.742,-69.375,-47.595,179.600,5.067,148.990
C07990=1120.737,-69.125,-47.605,179.601,5.073,148.991
C07991=1120.732,-68.875,-47.615,179.601,5.077,148.992
C07992=1120.726,-68.625,-47.626,179.601,5.083,148.993
C07993=1120.721,-68.375,-47.636,179.602,5.088,148.994
C07994=1120.715,-68.126,-47.646,179.602,5.093,148.996
C07995=1120.710,-67.877,-47.657,179.603,5.099,148.996
C07996=1120.706,-67.627,-47.667,179.602,5.104,148.998
C07997=1120.700,-67.377,-47.677,179.603,5.109,148.999
C07998=1120.695,-67.127,-47.688,179.603,5.115,149.000
C07999=1120.690,-66.877,-47.698,179.604,5.119,149.001
C08000=1120.684,-66.628,-47.708,179.605,5.125,149.002
C08001=1120.679,-66.378,-47.719,179.605,5.130,149.003
C08002=1120.674,-66.129,-47.730,179.606,5.136,149.004
C08003=1120.669,-65.878,-47.741,179.606,5.140,149.005
C08004=1120.663,-65.629,-47.751,179.606,5.146,149.006
C08005=1120.658,-65.379,-47.761,179.607,5.151,149.007
C08006=1120.653,-65.130,-47.772,179.607,5.156,149.008
C08007=1120.647,-64.880,-47.782,179.608,5.162,149.009
C08008=1120.642,-64.630,-47.793,179.608,5.167,149.010
C08009=1120.637,-64.380,-47.803,179.609,5.172,149.010
C08010=1120.631,-64.130,-47.815,179.609,5.177,149.011
C08011=1120.626,-63.881,-47.825,179.610,5.183,149.013
C08012=1120.621,-63.631,-47.836,179.610,5.188,149.013
C08013=1120.615,-63.381,-47.846,179.611,5.193,149.014
C08014=1120.610,-63.131,-47.857,179.612,5.198,149.015
C08015=1120.605,-62.882,-47.868,179.613,5.204,149.016
C08016=1120.600,-62.632,-47.878,179.613,5.208,149.017
C08017=1120.594,-62.383,-47.889,179.613,5.214,149.018
C08018=1120.589,-62.133,-47.900,179.614,5.220,149.019
C08019=1120.584,-61.883,-47.910,179.615,5.225,149.020
C08020=1120.580,-61.668,-47.920,179.616,5.229,149.021
C08021=1120.575,-61.453,-47.929,179.616,5.234,149.022
C08022=1120.570,-61.237,-47.938,179.617,5.238,149.022
C08023=1120.566,-61.022,-47.948,179.617,5.243,149.023
C08024=1120.561,-60.806,-47.957,179.618,5.247,149.024
C08025=1120.557,-60.591,-47.966,179.619,5.252,149.025
C08026=1120.553,-60.376,-47.976,179.620,5.256,149.026
C08027=1120.548,-60.161,-47.985,179.620,5.261,149.026
C08028=1120.542,-59.911,-47.995,179.620,5.265,149.027
C08029=1120.537,-59.661,-48.007,179.620,5.270,149.028
C08030=1120.531,-59.412,-48.017,179.619,5.274,149.030
C08031=1120.527,-59.162,-48.029,179.619,5.279,149.031
C08032=1120.521,-58.912,-48.039,179.619,5.283,149.032
C08033=1120.516,-58.663,-48.050,179.619,5.288,149.033
C08034=1120.511,-58.413,-48.061,179.619,5.294,149.034
C08035=1120.505,-58.163,-48.072,179.619,5.298,149.035
C08036=1120.500,-57.913,-48.083,179.619,5.303,149.036
C08037=1120.495,-57.664,-48.094,179.618,5.307,149.037
C08038=1120.490,-57.414,-48.104,179.618,5.312,149.038
C08039=1120.485,-57.164,-48.116,179.618,5.316,149.039
C08040=1120.479,-56.914,-48.126,179.618,5.321,149.040
C08041=1120.474,-56.665,-48.138,179.618,5.326,149.041
C08042=1120.469,-56.416,-48.149,179.617,5.330,149.042
C08043=1120.463,-56.165,-48.160,179.618,5.335,149.043
C08044=1120.459,-55.916,-48.171,179.617,5.339,149.045
C08045=1120.453,-55.666,-48.181,179.617,5.345,149.046
C08046=1120.448,-55.417,-48.193,179.617,5.349,149.047
C08047=1120.443,-55.166,-48.204,179.617,5.354,149.048
C08048=1120.437,-54.917,-48.215,179.617,5.359,149.049
C08049=1120.433,-54.667,-48.226,179.616,5.363,149.050
C08050=1120.428,-54.417,-48.237,179.616,5.368,149.051
C08051=1120.422,-54.168,-48.248,179.616,5.372,149.052
C08052=1120.417,-53.918,-48.259,179.616,5.377,149.053
C08053=1120.411,-53.669,-48.270,179.616,5.382,149.054
C08054=1120.406,-53.419,-48.281,179.615,5.386,149.055
C08055=1120.401,-53.169,-48.292,179.616,5.391,149.056
C08056=1120.396,-52.920,-48.303,179.615,5.396,149.057
C08057=1120.390,-52.670,-48.315,179.615,5.401,149.059
C08058=1120.385,-52.419,-48.325,179.615,5.405,149.059
C08059=1120.380,-52.171,-48.336,179.615,5.410,149.061
C08060=1120.375,-51.921,-48.348,179.614,5.415,149.062
C08061=1120.370,-51.671,-48.359,179.614,5.419,149.063
C08062=1120.364,-51.421,-48.370,179.614,5.424,149.064
C08063=1120.359,-51.172,-48.382,179.614,5.428,149.065
C08064=1120.354,-50.922,-48.393,179.614,5.433,149.066
C08065=1120.348,-50.672,-48.404,179.614,5.438,149.067
C08066=1120.343,-50.422,-48.415,179.613,5.443,149.068
C08067=1120.338,-50.173,-48.426,179.613,5.448,149.069
C08068=1120.333,-49.923,-48.438,179.613,5.452,149.070
C08069=1120.327,-49.673,-48.448,179.613,5.457,149.071
C08070=1120.322,-49.423,-48.460,179.613,5.462,149.073
C08071=1120.317,-49.174,-48.472,179.613,5.466,149.073
C08072=1120.312,-48.925,-48.482,179.613,5.471,149.075
C08073=1120.307,-48.675,-48.494,179.612,5.475,149.076
C08074=1120.302,-48.425,-48.505,179.612,5.480,149.077
C08075=1120.296,-48.175,-48.517,179.612,5.485,149.078
C08076=1120.292,-47.960,-48.527,179.612,5.489,149.079
C08077=1120.287,-47.744,-48.536,179.612,5.493,149.080
C08078=1120.283,-47.529,-48.546,179.612,5.497,149.081
C08079=1120.278,-47.314,-48.555,179.611,5.501,149.081
C08080=1120.274,-47.099,-48.565,179.611,5.505,149.083
C08081=1120.269,-46.884,-48.575,179.611,5.509,149.084
C08082=1120.265,-46.669,-48.585,179.610,5.513,149.084
C08083=1120.260,-46.454,-48.595,179.610,5.517,149.085
C08084=1120.255,-46.204,-48.607,179.611,5.522,149.086
C08085=1120.249,-45.954,-48.617,179.611,5.527,149.087
C08086=1120.244,-45.704,-48.629,179.610,5.531,149.089
C08087=1120.239,-45.455,-48.640,179.610,5.537,149.090
C08088=1120.234,-45.205,-48.652,179.610,5.541,149.091
C08089=1120.229,-44.956,-48.663,179.610,5.546,149.092
C08090=1120.223,-44.706,-48.675,179.610,5.551,149.093
C08091=1120.218,-44.456,-48.687,179.609,5.555,149.094
C08092=1120.213,-44.206,-48.698,179.609,5.560,149.095
C08093=1120.208,-43.957,-48.710,179.609,5.564,149.096
C08094=1120.202,-43.708,-48.721,179.609,5.569,149.097
C08095=1120.197,-43.458,-48.733,179.609,5.575,149.098
C08096=1120.192,-43.208,-48.744,179.608,5.578,149.099
C08097=1120.187,-42.958,-48.756,179.608,5.584,149.100
C08098=1120.182,-42.708,-48.766,179.611,5.590,149.101
C08099=1120.176,-42.459,-48.778,179.612,5.595,149.102
C08100=1120.171,-42.209,-48.789,179.613,5.600,149.103
C08101=1120.166,-41.959,-48.801,179.614,5.606,149.104
C08102=1120.160,-41.710,-48.814,179.616,5.611,149.104
C08103=1120.156,-41.460,-48.825,179.617,5.617,149.105
C08104=1120.150,-41.210,-48.837,179.618,5.622,149.106
C08105=1120.145,-40.961,-48.848,179.619,5.627,149.107
C08106=1120.140,-40.711,-48.860,179.621,5.632,149.107
C08107=1120.134,-40.461,-48.871,179.622,5.638,149.108
C08108=1120.130,-40.212,-48.883,179.623,5.643,149.109
C08109=1120.124,-39.962,-48.895,179.624,5.649,149.110
C08110=1120.119,-39.712,-48.906,179.626,5.654,149.110
C08111=1120.114,-39.462,-48.918,179.627,5.659,149.111
C08112=1120.109,-39.212,-48.930,179.628,5.664,149.112
C08113=1120.103,-38.964,-48.942,179.629,5.669,149.113
C08114=1120.098,-38.714,-48.953,179.630,5.674,149.114
C08115=1120.093,-38.464,-48.965,179.631,5.679,149.115
C08116=1120.087,-38.214,-48.977,179.631,5.684,149.115
C08117=1120.082,-37.964,-48.989,179.633,5.689,149.116
C08118=1120.077,-37.715,-49.001,179.633,5.694,149.117
C08119=1120.072,-37.465,-49.013,179.635,5.699,149.118
C08120=1120.067,-37.215,-49.025,179.635,5.704,149.119
C08121=1120.061,-36.965,-49.037,179.636,5.708,149.119
C08122=1120.057,-36.716,-49.049,179.637,5.714,149.120
C08123=1120.051,-36.467,-49.060,179.638,5.718,149.121
C08124=1120.046,-36.217,-49.072,179.639,5.723,149.122
C08125=1120.040,-35.967,-49.084,179.639,5.727,149.123
C08126=1120.036,-35.718,-49.096,179.640,5.732,149.124
C08127=1120.031,-35.468,-49.108,179.641,5.737,149.124
C08128=1120.025,-35.218,-49.120,179.641,5.741,149.125
C08129=1120.020,-34.969,-49.132,179.641,5.746,149.126
C08130=1120.014,-34.719,-49.144,179.642,5.750,149.127
C08131=1120.009,-34.469,-49.156,179.643,5.755,149.128
C08132=1120.005,-34.254,-49.167,179.643,5.759,149.128
C08133=1120.001,-34.039,-49.177,179.644,5.763,149.129
C08134=1119.996,-33.824,-49.188,179.644,5.767,149.130
C08135=1119.991,-33.609,-49.198,179.644,5.771,149.131
C08136=1119.987,-33.394,-49.209,179.644,5.774,149.131
C08137=1119.983,-33.179,-49.219,179.645,5.779,149.132
C08138=1119.978,-32.964,-49.229,179.645,5.782,149.133
C08139=1119.973,-32.749,-49.239,179.645,5.786,149.134
C08140=1119.968,-32.499,-49.252,179.645,5.790,149.135
C08141=1119.963,-32.249,-49.264,179.646,5.795,149.135
C08142=1119.958,-32.000,-49.275,179.646,5.800,149.136
C08143=1119.953,-31.750,-49.288,179.646,5.804,149.137
C08144=1119.948,-31.500,-49.300,179.646,5.808,149.138
C08145=1119.943,-31.250,-49.312,179.646,5.812,149.139
C08146=1119.937,-31.001,-49.324,179.646,5.816,149.140
C08147=1119.932,-30.751,-49.337,179.647,5.821,149.141
C08148=1119.927,-30.501,-49.349,179.646,5.825,149.142
C08149=1119.922,-30.252,-49.361,179.646,5.829,149.143
C08150=1119.916,-30.002,-49.373,179.646,5.834,149.144
C08151=1119.911,-29.753,-49.386,179.646,5.838,149.145
C08152=1119.906,-29.503,-49.398,179.646,5.842,149.146
C08153=1119.901,-29.254,-49.410,179.645,5.846,149.147
C08154=1119.896,-29.004,-49.422,179.645,5.850,149.148
C08155=1119.891,-28.755,-49.434,179.645,5.854,149.149
C08156=1119.885,-28.505,-49.446,179.644,5.858,149.150
C08157=1119.880,-28.255,-49.459,179.644,5.862,149.151
C08158=1119.875,-28.005,-49.471,179.644,5.867,149.152
C08159=1119.870,-27.755,-49.484,179.643,5.871,149.153
C08160=1119.865,-27.506,-49.496,179.643,5.875,149.154
C08161=1119.860,-27.256,-49.508,179.642,5.879,149.155
C08162=1119.855,-27.007,-49.521,179.642,5.884,149.156
C08163=1119.849,-26.757,-49.533,179.642,5.888,149.157
C08164=1119.844,-26.507,-49.545,179.641,5.892,149.158
C08165=1119.839,-26.258,-49.557,179.640,5.896,149.159
C08166=1119.834,-26.008,-49.570,179.639,5.900,149.160
C08167=1119.828,-25.759,-49.582,179.640,5.905,149.161
C08168=1119.824,-25.508,-49.595,179.640,5.909,149.162
C08169=1119.819,-25.259,-49.607,179.641,5.914,149.163
C08170=1119.813,-25.010,-49.620,179.642,5.920,149.164
C08171=1119.808,-24.760,-49.632,179.642,5.924,149.165
C08172=1119.803,-24.510,-49.644,179.643,5.929,149.166
C08173=1119.797,-24.260,-49.656,179.643,5.934,149.167
C08174=1119.792,-24.011,-49.669,179.644,5.939,149.168
C08175=1119.787,-23.762,-49.681,179.645,5.944,149.168
C08176=1119.782,-23.511,-49.694,179.645,5.949,149.169
C08177=1119.777,-23.262,-49.706,179.646,5.954,149.170
C08178=1119.772,-23.013,-49.719,179.646,5.958,149.171
C08179=1119.766,-22.763,-49.732,179.647,5.963,149.172
C08180=1119.761,-22.513,-49.744,179.647,5.967,149.173
C08181=1119.756,-22.264,-49.756,179.649,5.973,149.174
C08182=1119.751,-22.014,-49.769,179.649,5.978,149.174
C08183=1119.746,-21.764,-49.782,179.650,5.982,149.175
C08184=1119.741,-21.514,-49.794,179.650,5.987,149.176
C08185=1119.735,-21.265,-49.807,179.650,5.992,149.177
C08186=1119.730,-21.016,-49.819,179.651,5.997,149.178
C08187=1119.726,-20.766,-49.832,179.652,6.001,149.179
C08188=1119.721,-20.551,-49.843,179.652,6.006,149.180
C08189=1119.716,-20.336,-49.854,179.653,6.009,149.180
C08190=1119.712,-20.120,-49.864,179.654,6.014,149.181
C08191=1119.707,-19.906,-49.876,179.654,6.018,149.182
C08192=1119.702,-19.691,-49.886,179.655,6.022,149.183
C08193=1119.699,-19.476,-49.897,179.656,6.026,149.183
C08194=1119.694,-19.261,-49.908,179.656,6.030,149.184
C08195=1119.690,-19.045,-49.920,179.656,6.034,149.185
C08196=1119.685,-18.796,-49.932,179.657,6.039,149.185
C08197=1119.679,-18.547,-49.945,179.658,6.043,149.186
C08198=1119.674,-18.297,-49.957,179.658,6.048,149.187
C08199=1119.669,-18.046,-49.970,179.659,6.053,149.188
C08200=1119.664,-17.797,-49.983,179.659,6.058,149.189
C08201=1119.659,-17.548,-49.995,179.660,6.062,149.190
C08202=1119.653,-17.298,-50.008,179.661,6.067,149.191
C08203=1119.648,-17.048,-50.022,179.661,6.071,149.191
C08204=1119.643,-16.799,-50.034,179.662,6.076,149.192
C08205=1119.638,-16.549,-50.047,179.663,6.081,149.193
C08206=1119.633,-16.300,-50.059,179.663,6.085,149.194
C08207=1119.628,-16.050,-50.073,179.664,6.090,149.195
C08208=1119.622,-15.800,-50.086,179.664,6.095,149.196
C08209=1119.617,-15.551,-50.098,179.665,6.099,149.196
C08210=1119.613,-15.301,-50.111,179.666,6.105,149.197
C08211=1119.607,-15.052,-50.124,179.667,6.109,149.198
C08212=1119.602,-14.802,-50.137,179.667,6.114,149.199
C08213=1119.597,-14.552,-50.150,179.668,6.118,149.200
C08214=1119.591,-14.303,-50.163,179.669,6.123,149.201
C08215=1119.586,-14.053,-50.176,179.669,6.128,149.201
C08216=1119.582,-13.803,-50.189,179.670,6.133,149.202
C08217=1119.576,-13.554,-50.202,179.671,6.137,149.203
C08218=1119.571,-13.304,-50.215,179.671,6.142,149.204
C08219=1119.567,-13.055,-50.228,179.672,6.146,149.205
C08220=1119.561,-12.805,-50.241,179.673,6.151,149.205
C08221=1119.556,-12.556,-50.254,179.673,6.155,149.206
C08222=1119.551,-12.306,-50.267,179.674,6.160,149.207
C08223=1119.545,-12.056,-50.280,179.674,6.165,149.208
C08224=1119.540,-11.807,-50.293,179.675,6.169,149.209
C08225=1119.535,-11.557,-50.306,179.676,6.174,149.210
C08226=1119.530,-11.308,-50.320,179.676,6.178,149.211
C08227=1119.525,-11.058,-50.333,179.677,6.182,149.211
C08228=1119.520,-10.808,-50.346,179.677,6.187,149.212
C08229=1119.514,-10.559,-50.358,179.678,6.192,149.213
C08230=1119.509,-10.309,-50.372,179.679,6.196,149.214
C08231=1119.504,-10.060,-50.385,179.679,6.201,149.215
C08232=1119.500,-9.810,-50.398,179.680,6.206,149.215
C08233=1119.494,-9.560,-50.411,179.680,6.210,149.216
C08234=1119.489,-9.310,-50.424,179.681,6.215,149.217
C08235=1119.484,-9.061,-50.438,179.682,6.219,149.218
C08236=1119.479,-8.812,-50.451,179.682,6.224,149.219
C08237=1119.474,-8.562,-50.464,179.683,6.228,149.219
C08238=1119.468,-8.312,-50.477,179.684,6.233,149.220
C08239=1119.463,-8.063,-50.491,179.684,6.238,149.221
C08240=1119.458,-7.813,-50.504,179.685,6.242,149.222
C08241=1119.453,-7.563,-50.518,179.686,6.247,149.223
C08242=1119.448,-7.314,-50.531,179.686,6.252,149.224
C08243=1119.443,-7.064,-50.544,179.687,6.256,149.224
C08244=1119.438,-6.849,-50.556,179.687,6.260,149.225
C08245=1119.434,-6.634,-50.567,179.687,6.263,149.226
C08246=1119.429,-6.420,-50.579,179.688,6.268,149.227
C08247=1119.425,-6.204,-50.590,179.689,6.271,149.227
C08248=1119.421,-5.990,-50.601,179.689,6.275,149.228
C08249=1119.417,-5.775,-50.613,179.690,6.280,149.229
C08250=1119.412,-5.560,-50.624,179.690,6.283,149.229
C08251=1119.408,-5.345,-50.636,179.691,6.287,149.230
C08252=1119.402,-5.095,-50.649,179.691,6.291,149.231
C08253=1119.397,-4.846,-50.663,179.692,6.296,149.232
C08254=1119.392,-4.596,-50.676,179.693,6.300,149.233
C08255=1119.387,-4.347,-50.690,179.693,6.305,149.233
C08256=1119.382,-4.097,-50.703,179.694,6.310,149.234
C08257=1119.377,-3.848,-50.717,179.695,6.314,149.235
C08258=1119.372,-3.598,-50.730,179.695,6.319,149.236
C08259=1119.367,-3.348,-50.743,179.696,6.323,149.237
C08260=1119.362,-3.098,-50.757,179.697,6.328,149.237
C08261=1119.357,-2.849,-50.770,179.697,6.332,149.238
C08262=1119.352,-2.599,-50.784,179.697,6.337,149.239
C08263=1119.346,-2.350,-50.798,179.698,6.341,149.240
C08264=1119.341,-2.100,-50.811,179.699,6.346,149.241
C08265=1119.336,-1.851,-50.824,179.699,6.350,149.242
C08266=1119.331,-1.601,-50.839,179.700,6.355,149.242
C08267=1119.326,-1.352,-50.852,179.701,6.359,149.243
C08268=1119.321,-1.102,-50.866,179.701,6.364,149.244
C08269=1119.316,-0.852,-50.880,179.702,6.369,149.245
C08270=1119.310,-0.603,-50.892,179.702,6.372,149.246
C08271=1119.306,-0.353,-50.907,179.703,6.377,149.247
C08272=1119.300,-0.103,-50.920,179.703,6.382,149.247
C08273=1119.295,0.146,-50.934,179.704,6.387,149.248
C08274=1119.290,0.395,-50.948,179.705,6.391,149.249
C08275=1119.285,0.645,-50.961,179.705,6.396,149.250
C08276=1119.280,0.895,-50.975,179.706,6.400,149.251
C08277=1119.275,1.144,-50.989,179.706,6.404,149.252
C08278=1119.270,1.394,-51.002,179.707,6.409,149.252
C08279=1119.264,1.643,-51.016,179.707,6.413,149.253
C08280=1119.259,1.893,-51.030,179.708,6.418,149.254
C08281=1119.255,2.143,-51.043,179.708,6.423,149.255
C08282=1119.249,2.392,-51.057,179.709,6.427,149.256
C08283=1119.244,2.642,-51.072,179.710,6.432,149.256
C08284=1119.239,2.892,-51.085,179.710,6.436,149.257
C08285=1119.234,3.141,-51.098,179.710,6.440,149.258
C08286=1119.229,3.390,-51.113,179.711,6.445,149.259
C08287=1119.224,3.641,-51.126,179.712,6.450,149.260
C08288=1119.218,3.890,-51.140,179.712,6.454,149.261
C08289=1119.213,4.139,-51.154,179.713,6.459,149.262
C08290=1119.209,4.389,-51.168,179.713,6.464,149.262
C08291=1119.203,4.638,-51.182,179.713,6.468,149.263
C08292=1119.198,4.888,-51.196,179.714,6.472,149.264
C08293=1119.193,5.138,-51.210,179.715,6.477,149.265
C08294=1119.188,5.387,-51.224,179.715,6.481,149.266
C08295=1119.184,5.636,-51.237,179.716,6.486,149.267
C08296=1119.179,5.886,-51.252,179.717,6.491,149.268
C08297=1119.173,6.136,-51.265,179.717,6.496,149.268
C08298=1119.168,6.385,-51.279,179.717,6.499,149.269
C08299=1119.163,6.635,-51.294,179.718,6.504,149.270
C08300=1119.158,6.849,-51.305,179.719,6.508,149.271
C08301=1119.154,7.064,-51.317,179.719,6.512,149.271
C08302=1119.149,7.280,-51.330,179.719,6.516,149.272
C08303=1119.145,7.494,-51.342,179.720,6.520,149.273
C08304=1119.141,7.709,-51.353,179.720,6.524,149.274
C08305=1119.137,7.924,-51.366,179.721,6.527,149.274
C08306=1119.132,8.139,-51.378,179.721,6.531,149.275
C08307=1119.127,8.353,-51.390,179.722,6.536,149.276
C08308=1119.122,8.603,-51.404,179.722,6.540,149.277
C08309=1119.117,8.852,-51.418,179.723,6.545,149.278
C08310=1119.112,9.102,-51.433,179.724,6.549,149.278
C08311=1119.107,9.351,-51.447,179.724,6.554,149.279
C08312=1119.102,9.601,-51.461,179.725,6.559,149.280
C08313=1119.097,9.851,-51.475,179.725,6.564,149.281
C08314=1119.092,10.101,-51.489,179.726,6.568,149.282
C08315=1119.086,10.350,-51.503,179.727,6.573,149.282
C08316=1119.081,10.600,-51.517,179.728,6.577,149.283
C08317=1119.076,10.849,-51.531,179.729,6.582,149.284
C08318=1119.072,11.098,-51.546,179.729,6.586,149.285
C08319=1119.067,11.348,-51.561,179.730,6.591,149.286
C08320=1119.061,11.597,-51.574,179.731,6.595,149.286
C08321=1119.056,11.847,-51.589,179.731,6.600,149.287
C08322=1119.051,12.097,-51.603,179.732,6.605,149.288
C08323=1119.046,12.346,-51.617,179.733,6.609,149.289
C08324=1119.041,12.596,-51.632,179.733,6.614,149.290
C08325=1119.036,12.845,-51.645,179.734,6.618,149.291
C08326=1119.031,13.095,-51.660,179.735,6.623,149.291
C08327=1119.026,13.344,-51.674,179.736,6.628,149.292
C08328=1119.021,13.594,-51.688,179.737,6.632,149.293
C08329=1119.016,13.844,-51.703,179.737,6.637,149.294
C08330=1119.011,14.094,-51.717,179.738,6.641,149.295
C08331=1119.006,14.342,-51.731,179.739,6.646,149.295
C08332=1119.001,14.592,-51.746,179.739,6.650,149.296
C08333=1118.996,14.841,-51.760,179.740,6.655,149.297
C08334=1118.991,15.091,-51.774,179.741,6.659,149.298
C08335=1118.986,15.341,-51.789,179.742,6.664,149.298
C08336=1118.981,15.590,-51.804,179.742,6.668,149.299
C08337=1118.976,15.840,-51.818,179.743,6.673,149.300
C08338=1118.970,16.089,-51.832,179.744,6.677,149.301
C08339=1118.965,16.339,-51.847,179.745,6.682,149.301
C08340=1118.960,16.588,-51.861,179.746,6.686,149.302
C08341=1118.955,16.837,-51.876,179.747,6.691,149.303
C08342=1118.951,17.087,-51.890,179.747,6.695,149.304
C08343=1118.945,17.337,-51.905,179.748,6.700,149.304
C08344=1118.940,17.587,-51.919,179.749,6.704,149.305
C08345=1118.935,17.836,-51.934,179.750,6.709,149.306
C08346=1118.930,18.086,-51.949,179.750,6.714,149.307
C08347=1118.925,18.335,-51.963,179.751,6.718,149.307
C08348=1118.919,18.584,-51.978,179.752,6.723,149.308
C08349=1118.914,18.834,-51.992,179.753,6.727,149.309
C08350=1118.909,19.084,-52.007,179.754,6.731,149.310
C08351=1118.905,19.333,-52.022,179.755,6.736,149.311
C08352=1118.900,19.582,-52.036,179.756,6.740,149.311
C08353=1118.894,19.832,-52.051,179.756,6.745,149.312
C08354=1118.889,20.081,-52.066,179.757,6.749,149.313
C08355=1118.885,20.331,-52.080,179.758,6.754,149.313
C08356=1118.880,20.546,-52.093,179.759,6.757,149.314
C08357=1118.876,20.761,-52.105,179.760,6.761,149.315
C08358=1118.871,20.976,-52.118,179.760,6.765,149.315
C08359=1118.868,21.190,-52.131,179.761,6.768,149.316
C08360=1118.863,21.405,-52.144,179.762,6.773,149.317
C08361=1118.858,21.620,-52.156,179.762,6.776,149.317
C08362=1118.854,21.834,-52.169,179.764,6.780,149.318
C08363=1118.849,22.049,-52.182,179.764,6.784,149.318
C08364=1118.844,22.299,-52.196,179.765,6.788,149.319
C08365=1118.840,22.548,-52.211,179.766,6.793,149.320
C08366=1118.834,22.798,-52.226,179.767,6.797,149.321
C08367=1118.829,23.047,-52.241,179.768,6.801,149.321
C08368=1118.824,23.297,-52.255,179.768,6.806,149.322
C08369=1118.819,23.546,-52.271,179.769,6.810,149.323
C08370=1118.814,23.796,-52.285,179.771,6.815,149.323
C08371=1118.809,24.045,-52.300,179.772,6.819,149.324
C08372=1118.804,24.294,-52.316,179.772,6.824,149.325
C08373=1118.799,24.544,-52.330,179.773,6.828,149.326
C08374=1118.794,24.793,-52.345,179.774,6.832,149.326
C08375=1118.789,25.043,-52.360,179.775,6.836,149.327
C08376=1118.785,25.293,-52.375,179.775,6.841,149.328
C08377=1118.779,25.543,-52.390,179.776,6.845,149.328
C08378=1118.774,25.792,-52.405,179.777,6.849,149.329
C08379=1118.770,26.041,-52.420,179.778,6.854,149.330
C08380=1118.764,26.291,-52.435,179.779,6.858,149.330
C08381=1118.759,26.540,-52.450,179.780,6.863,149.331
C08382=1118.754,26.790,-52.466,179.781,6.867,149.332
C08383=1118.749,27.039,-52.480,179.782,6.871,149.333
C08384=1118.744,27.289,-52.495,179.783,6.876,149.333
C08385=1118.739,27.538,-52.510,179.784,6.880,149.334
C08386=1118.734,27.788,-52.525,179.785,6.884,149.335
C08387=1118.729,28.037,-52.540,179.786,6.888,149.335
C08388=1118.724,28.286,-52.555,179.787,6.893,149.336
C08389=1118.719,28.537,-52.570,179.788,6.898,149.337
C08390=1118.714,28.786,-52.585,179.788,6.901,149.337
C08391=1118.709,29.035,-52.601,179.789,6.905,149.338
C08392=1118.704,29.284,-52.616,179.791,6.910,149.339
C08393=1118.699,29.534,-52.631,179.792,6.914,149.339
C08394=1118.694,29.784,-52.646,179.793,6.918,149.340
C08395=1118.688,30.033,-52.662,179.794,6.923,149.341
C08396=1118.684,30.282,-52.676,179.795,6.927,149.341
C08397=1118.679,30.533,-52.692,179.796,6.931,149.342
C08398=1118.673,30.782,-52.707,179.797,6.936,149.343
C08399=1118.669,31.031,-52.722,179.798,6.940,149.343
C08400=1118.663,31.281,-52.738,179.799,6.945,149.344
C08401=1118.659,31.530,-52.753,179.800,6.949,149.345
C08402=1118.653,31.779,-52.768,179.800,6.952,149.345
C08403=1118.649,32.030,-52.783,179.801,6.957,149.346
C08404=1118.644,32.279,-52.799,179.802,6.961,149.347
C08405=1118.639,32.528,-52.814,179.803,6.965,149.347
C08406=1118.634,32.777,-52.829,179.804,6.970,149.348
C08407=1118.628,33.027,-52.845,179.805,6.974,149.349
C08408=1118.624,33.277,-52.860,179.806,6.978,149.349
C08409=1118.619,33.526,-52.876,179.807,6.983,149.350
C08410=1118.613,33.775,-52.891,179.809,6.987,149.351
C08411=1118.609,34.025,-52.906,179.810,6.991,149.351
C08412=1118.604,34.239,-52.919,179.811,6.994,149.352
C08413=1118.600,34.454,-52.933,179.811,6.998,149.352
C08414=1118.595,34.669,-52.946,179.813,7.002,149.353
C08415=1118.591,34.883,-52.960,179.813,7.005,149.353
C08416=1118.587,35.099,-52.973,179.814,7.009,149.354
C08417=1118.583,35.313,-52.986,179.815,7.013,149.355
C08418=1118.579,35.528,-52.999,179.816,7.016,149.355
C08419=1118.574,35.742,-53.013,179.817,7.020,149.356
C08420=1118.569,35.991,-53.029,179.817,7.024,149.356
C08421=1118.564,36.241,-53.044,179.818,7.028,149.357
C08422=1118.560,36.491,-53.060,179.820,7.032,149.357
C08423=1118.554,36.740,-53.075,179.821,7.036,149.358
C08424=1118.549,36.989,-53.091,179.822,7.041,149.359
C08425=1118.543,37.239,-53.106,179.823,7.045,149.359
C08426=1118.539,37.489,-53.122,179.824,7.049,149.360
C08427=1118.534,37.738,-53.137,179.825,7.053,149.361
C08428=1118.529,37.987,-53.153,179.826,7.058,149.361
C08429=1118.523,38.237,-53.168,179.827,7.062,149.362
C08430=1118.519,38.487,-53.184,179.829,7.066,149.362
C08431=1118.514,38.735,-53.200,179.829,7.070,149.363
C08432=1118.509,38.985,-53.216,179.831,7.074,149.364
C08433=1118.504,39.235,-53.232,179.832,7.078,149.364
C08434=1118.499,39.484,-53.247,179.833,7.082,149.365
C08435=1118.494,39.733,-53.262,179.834,7.087,149.366
C08436=1118.489,39.984,-53.278,179.835,7.091,149.366
C08437=1118.484,40.232,-53.294,179.836,7.095,149.367
C08438=1118.479,40.482,-53.310,179.837,7.099,149.367
C08439=1118.474,40.732,-53.326,179.838,7.104,149.368
C08440=1118.469,40.981,-53.341,179.839,7.107,149.369
C08441=1118.464,41.230,-53.357,179.840,7.111,149.369
C08442=1118.459,41.480,-53.373,179.842,7.115,149.370
C08443=1118.454,41.729,-53.389,179.843,7.120,149.370
C08444=1118.449,41.979,-53.404,179.844,7.124,149.371
C08445=1118.444,42.228,-53.421,179.845,7.128,149.372
C08446=1118.439,42.477,-53.437,179.846,7.132,149.372
C08447=1118.435,42.727,-53.452,179.847,7.136,149.373
C08448=1118.429,42.977,-53.468,179.848,7.141,149.373
C08449=1118.424,43.225,-53.484,179.850,7.145,149.374
C08450=1118.419,43.476,-53.500,179.850,7.148,149.374
C08451=1118.414,43.725,-53.515,179.852,7.153,149.375
C08452=1118.409,43.974,-53.532,179.853,7.157,149.376
C08453=1118.404,44.224,-53.548,179.854,7.161,149.376
C08454=1118.399,44.473,-53.563,179.855,7.165,149.377
C08455=1118.394,44.723,-53.580,179.856,7.169,149.377
C08456=1118.389,44.972,-53.596,179.857,7.174,149.378
C08457=1118.384,45.222,-53.612,179.859,7.178,149.379
C08458=1118.379,45.471,-53.628,179.860,7.182,149.379
C08459=1118.374,45.720,-53.643,179.861,7.185,149.380
C08460=1118.369,45.970,-53.660,179.862,7.189,149.380
C08461=1118.364,46.219,-53.676,179.863,7.194,149.381
C08462=1118.359,46.469,-53.692,179.864,7.198,149.382
C08463=1118.355,46.718,-53.707,179.866,7.202,149.382
C08464=1118.350,46.967,-53.724,179.867,7.206,149.383
C08465=1118.344,47.217,-53.740,179.868,7.210,149.383
C08466=1118.340,47.467,-53.757,179.869,7.214,149.384
C08467=1118.334,47.716,-53.772,179.871,7.219,149.384
C08468=1118.330,47.930,-53.786,179.871,7.222,149.385
C08469=1118.326,48.145,-53.800,179.872,7.225,149.385
C08470=1118.322,48.360,-53.814,179.874,7.229,149.386
C08471=1118.318,48.574,-53.828,179.874,7.232,149.386
C08472=1118.313,48.788,-53.841,179.875,7.235,149.387
C08473=1118.309,49.004,-53.856,179.877,7.239,149.387
C08474=1118.305,49.218,-53.870,179.877,7.243,149.388
C08475=1118.300,49.432,-53.883,179.878,7.246,149.388
C08476=1118.296,49.682,-53.900,179.879,7.250,149.389
C08477=1118.291,49.931,-53.916,179.881,7.254,149.389
C08478=1118.286,50.181,-53.932,179.882,7.259,149.390
C08479=1118.281,50.429,-53.949,179.884,7.262,149.390
C08480=1118.276,50.680,-53.965,179.885,7.267,149.391
C08481=1118.271,50.929,-53.982,179.886,7.271,149.392
C08482=1118.266,51.178,-53.998,179.887,7.274,149.392
C08483=1118.261,51.428,-54.014,179.888,7.278,149.393
C08484=1118.256,51.677,-54.030,179.889,7.282,149.393
C08485=1118.251,51.927,-54.047,179.890,7.287,149.394
C08486=1118.246,52.176,-54.063,179.892,7.291,149.394
C08487=1118.242,52.425,-54.079,179.893,7.295,149.395
C08488=1118.236,52.675,-54.096,179.894,7.299,149.396
C08489=1118.231,52.924,-54.113,179.896,7.303,149.396
C08490=1118.226,53.173,-54.129,179.897,7.307,149.397
C08491=1118.221,53.423,-54.145,179.898,7.311,149.397
C08492=1118.217,53.672,-54.162,179.899,7.315,149.398
C08493=1118.211,53.921,-54.179,179.900,7.319,149.398
C08494=1118.206,54.172,-54.195,179.901,7.323,149.399
C08495=1118.201,54.420,-54.211,179.903,7.327,149.399
C08496=1118.197,54.670,-54.228,179.904,7.331,149.400
C08497=1118.191,54.920,-54.245,179.906,7.335,149.400
C08498=1118.186,55.168,-54.261,179.907,7.339,149.401
C08499=1118.182,55.419,-54.277,179.908,7.343,149.401
C08500=1118.177,55.667,-54.293,179.909,7.347,149.402
C08501=1118.171,55.917,-54.311,179.910,7.351,149.403
C08502=1118.167,56.167,-54.327,179.911,7.355,149.403
C08503=1118.162,56.415,-54.344,179.913,7.359,149.404
C08504=1118.157,56.665,-54.360,179.914,7.363,149.404
C08505=1118.152,56.915,-54.378,179.916,7.367,149.405
C08506=1118.147,57.164,-54.393,179.917,7.371,149.405
C08507=1118.142,57.414,-54.410,179.918,7.375,149.406
C08508=1118.137,57.663,-54.427,179.919,7.380,149.406
C08509=1118.132,57.912,-54.443,179.921,7.384,149.407
C08510=1118.127,58.162,-54.460,179.921,7.387,149.407
C08511=1118.122,58.411,-54.477,179.923,7.391,149.408
C08512=1118.117,58.660,-54.494,179.925,7.395,149.408
C08513=1118.113,58.910,-54.510,179.926,7.399,149.409
C08514=1118.107,59.159,-54.528,179.927,7.403,149.409
C08515=1118.102,59.408,-54.544,179.928,7.407,149.410
C08516=1118.097,59.658,-54.561,179.930,7.411,149.411
C08517=1118.093,59.908,-54.578,179.931,7.416,149.411
C08518=1118.088,60.157,-54.595,179.933,7.420,149.412
C08519=1118.082,60.406,-54.611,179.934,7.423,149.412
C08520=1118.078,60.656,-54.628,179.935,7.427,149.413
C08521=1118.073,60.905,-54.645,179.936,7.431,149.413
C08522=1118.068,61.154,-54.662,179.937,7.435,149.414
C08523=1118.063,61.404,-54.678,179.939,7.439,149.414
C08524=1118.059,61.618,-54.694,179.940,7.442,149.415
C08525=1118.055,61.833,-54.707,179.941,7.446,149.415
C08526=1118.051,62.047,-54.723,179.942,7.449,149.415
C08527=1118.047,62.261,-54.737,179.943,7.452,149.416
C08528=1118.042,62.476,-54.752,179.945,7.456,149.416
C08529=1118.038,62.690,-54.766,179.945,7.460,149.417
C08530=1118.033,62.905,-54.781,179.947,7.464,149.417
C08531=1118.030,63.119,-54.795,179.948,7.467,149.418
C08532=1118.024,63.369,-54.813,179.949,7.471,149.418
C08533=1118.020,63.618,-54.829,179.951,7.475,149.419
C08534=1118.014,63.868,-54.846,179.952,7.479,149.419
C08535=1118.010,64.117,-54.863,179.954,7.483,149.420
C08536=1118.005,64.366,-54.881,179.954,7.486,149.420
C08537=1118.000,64.616,-54.898,179.956,7.490,149.421
C08538=1117.995,64.866,-54.915,179.957,7.494,149.421
C08539=1117.990,65.114,-54.931,179.958,7.498,149.422
C08540=1117.985,65.363,-54.949,179.960,7.502,149.422
C08541=1117.980,65.613,-54.966,179.961,7.506,149.423
C08542=1117.975,65.863,-54.983,179.963,7.511,149.423
C08543=1117.970,66.113,-55.000,179.964,7.514,149.424
C08544=1117.965,66.361,-55.017,179.966,7.518,149.424
C08545=1117.960,66.611,-55.035,179.967,7.523,149.425
C08546=1117.956,66.860,-55.051,179.968,7.527,149.425
C08547=1117.951,67.109,-55.069,179.969,7.530,149.426
C08548=1117.946,67.359,-55.087,179.970,7.534,149.426
C08549=1117.941,67.608,-55.103,179.972,7.538,149.427
C08550=1117.936,67.858,-55.121,179.974,7.542,149.427
C08551=1117.931,68.106,-55.138,179.975,7.546,149.428
C08552=1117.926,68.356,-55.155,179.976,7.550,149.428
C08553=1117.921,68.605,-55.173,179.978,7.554,149.429
C08554=1117.916,68.855,-55.189,179.979,7.558,149.429
C08555=1117.912,69.104,-55.207,179.981,7.562,149.430
C08556=1117.906,69.354,-55.225,179.982,7.566,149.430
C08557=1117.902,69.603,-55.242,179.983,7.570,149.431
C08558=1117.897,69.853,-55.259,179.985,7.574,149.431
C08559=1117.892,70.102,-55.277,179.986,7.577,149.432
C08560=1117.888,70.351,-55.294,179.987,7.582,149.432
C08561=1117.882,70.600,-55.312,179.988,7.585,149.433
C08562=1117.877,70.849,-55.329,179.990,7.589,149.433
C08563=1117.873,71.098,-55.346,179.992,7.593,149.434
C08564=1117.867,71.348,-55.363,179.993,7.598,149.434
C08565=1117.863,71.597,-55.381,179.994,7.601,149.435
C08566=1117.857,71.847,-55.399,179.996,7.605,149.435
C08567=1117.853,72.096,-55.416,179.997,7.610,149.436
C08568=1117.848,72.346,-55.433,179.999,7.614,149.436
C08569=1117.843,72.595,-55.451,-180.000,7.617,149.437
C08570=1117.838,72.845,-55.469,-179.998,7.621,149.437
C08571=1117.834,73.094,-55.486,-179.997,7.626,149.438
C08572=1117.829,73.343,-55.504,-179.996,7.630,149.438
C08573=1117.824,73.593,-55.521,-179.995,7.633,149.439
C08574=1117.819,73.842,-55.539,-179.994,7.637,149.439
C08575=1117.813,74.092,-55.556,-179.992,7.641,149.440
C08576=1117.809,74.340,-55.574,-179.990,7.645,149.440
C08577=1117.804,74.590,-55.592,-179.989,7.649,149.441
C08578=1117.799,74.839,-55.609,-179.988,7.653,149.441
C08579=1117.794,75.089,-55.627,-179.986,7.657,149.442
C08580=1117.789,75.303,-55.642,-179.985,7.660,149.442
C08581=1117.785,75.517,-55.658,-179.984,7.664,149.443
C08582=1117.782,75.732,-55.672,-179.983,7.667,149.443
C08583=1117.777,75.946,-55.687,-179.981,7.671,149.443
C08584=1117.773,76.160,-55.703,-179.980,7.674,149.444
C08585=1117.769,76.375,-55.718,-179.979,7.677,149.444
C08586=1117.765,76.589,-55.734,-179.977,7.681,149.445
C08587=1117.760,76.803,-55.749,-179.976,7.684,149.445
C08588=1117.755,77.053,-55.766,-179.975,7.688,149.446
C08589=1117.751,77.302,-55.784,-179.975,7.691,149.446
C08590=1117.746,77.551,-55.802,-179.973,7.695,149.447
C08591=1117.741,77.800,-55.820,-179.972,7.699,149.447
C08592=1117.736,78.049,-55.838,-179.971,7.702,149.448
C08593=1117.731,78.299,-55.855,-179.970,7.706,149.448
C08594=1117.727,78.549,-55.873,-179.969,7.709,149.449
C08595=1117.722,78.798,-55.891,-179.968,7.714,149.450
C08596=1117.717,79.047,-55.909,-179.967,7.717,149.450
C08597=1117.712,79.297,-55.927,-179.966,7.721,149.451
C08598=1117.707,79.546,-55.945,-179.966,7.725,149.451
C08599=1117.702,79.796,-55.963,-179.964,7.728,149.452
C08600=1117.697,80.045,-55.981,-179.964,7.732,149.452
C08601=1117.692,80.294,-55.999,-179.962,7.736,149.453
C08602=1117.687,80.543,-56.017,-179.961,7.740,149.453
C08603=1117.682,80.792,-56.035,-179.960,7.743,149.454
C08604=1117.677,81.041,-56.052,-179.959,7.748,149.454
C08605=1117.673,81.291,-56.071,-179.958,7.751,149.455
C08606=1117.668,81.541,-56.089,-179.957,7.755,149.456
C08607=1117.663,81.790,-56.107,-179.956,7.758,149.456
C08608=1117.658,82.039,-56.125,-179.955,7.762,149.457
C08609=1117.653,82.288,-56.143,-179.953,7.766,149.457
C08610=1117.648,82.537,-56.161,-179.953,7.770,149.458
C08611=1117.644,82.786,-56.179,-179.951,7.774,149.458
C08612=1117.639,83.036,-56.197,-179.950,7.777,149.459
C08613=1117.634,83.285,-56.215,-179.949,7.781,149.459
C08614=1117.629,83.535,-56.233,-179.947,7.785,149.460
C08615=1117.624,83.784,-56.251,-179.947,7.788,149.460
C08616=1117.620,84.033,-56.269,-179.945,7.792,149.461
C08617=1117.615,84.282,-56.287,-179.944,7.797,149.461
C08618=1117.610,84.531,-56.305,-179.943,7.800,149.462
C08619=1117.605,84.781,-56.323,-179.941,7.804,149.462
C08620=1117.600,85.031,-56.342,-179.940,7.808,149.463
C08621=1117.595,85.280,-56.360,-179.939,7.811,149.463
C08622=1117.590,85.529,-56.378,-179.938,7.815,149.464
C08623=1117.585,85.778,-56.396,-179.937,7.819,149.464
C08624=1117.581,86.028,-56.414,-179.936,7.822,149.465
C08625=1117.576,86.277,-56.432,-179.935,7.827,149.465
C08626=1117.571,86.526,-56.450,-179.933,7.830,149.466
C08627=1117.566,86.775,-56.469,-179.931,7.834,149.466
C08628=1117.561,87.024,-56.487,-179.931,7.838,149.467
C08629=1117.556,87.274,-56.506,-179.929,7.842,149.467
C08630=1117.551,87.524,-56.524,-179.928,7.846,149.468
C08631=1117.547,87.773,-56.542,-179.927,7.850,149.468
C08632=1117.542,88.022,-56.560,-179.926,7.853,149.469
C08633=1117.538,88.271,-56.579,-179.924,7.857,149.469
C08634=1117.532,88.521,-56.597,-179.923,7.861,149.470
C08635=1117.527,88.770,-56.615,-179.921,7.865,149.470
C08636=1117.523,88.984,-56.631,-179.920,7.868,149.471
C08637=1117.519,89.199,-56.647,-179.919,7.871,149.471
C08638=1117.515,89.413,-56.663,-179.918,7.875,149.472
C08639=1117.511,89.627,-56.678,-179.917,7.878,149.472
C08640=1117.506,89.841,-56.695,-179.915,7.881,149.472
C08641=1117.502,90.056,-56.710,-179.914,7.884,149.473
C08642=1117.498,90.270,-56.726,-179.913,7.888,149.473
C08643=1117.494,90.484,-56.742,-179.912,7.891,149.474
C08644=1117.489,90.733,-56.760,-179.910,7.895,149.474
C08645=1117.484,90.983,-56.779,-179.909,7.899,149.475
C08646=1117.480,91.232,-56.798,-179.907,7.903,149.475
C08647=1117.475,91.481,-56.816,-179.906,7.906,149.476
C08648=1117.469,91.731,-56.834,-179.905,7.910,149.476
C08649=1117.465,91.980,-56.853,-179.903,7.914,149.476
C08650=1117.460,92.229,-56.871,-179.902,7.918,149.477
C08651=1117.455,92.478,-56.889,-179.900,7.922,149.477
C08652=1117.451,92.728,-56.909,-179.899,7.926,149.478
C08653=1117.446,92.977,-56.927,-179.897,7.930,149.478
C08654=1117.441,93.226,-56.946,-179.896,7.934,149.479
C08655=1117.436,93.476,-56.965,-179.894,7.938,149.479
C08656=1117.431,93.725,-56.983,-179.893,7.941,149.480
C08657=1117.426,93.974,-57.002,-179.892,7.945,149.480
C08658=1117.421,94.224,-57.020,-179.890,7.949,149.481
C08659=1117.417,94.472,-57.039,-179.888,7.953,149.481
C08660=1117.412,94.720,-57.057,-179.887,7.956,149.481
C08661=1117.407,94.967,-57.076,-179.885,7.960,149.482
C08662=1117.403,95.214,-57.095,-179.884,7.964,149.482
C08663=1117.397,95.462,-57.113,-179.882,7.968,149.483
C08664=1117.392,95.709,-57.132,-179.880,7.972,149.483
C08665=1117.387,95.957,-57.150,-179.879,7.976,149.484
C08666=1117.383,96.204,-57.169,-179.877,7.980,149.484
C08667=1117.378,96.451,-57.188,-179.876,7.984,149.484
C08668=1117.373,96.701,-57.207,-179.874,7.988,149.485
C08669=1117.369,96.950,-57.226,-179.872,7.991,149.485
C08670=1117.364,97.200,-57.244,-179.870,7.995,149.486
C08671=1117.359,97.449,-57.263,-179.869,7.999,149.486
C08672=1117.354,97.697,-57.282,-179.867,8.003,149.486
C08673=1117.349,97.947,-57.301,-179.866,8.007,149.487
C08674=1117.345,98.196,-57.320,-179.864,8.011,149.487
C08675=1117.340,98.446,-57.338,-179.862,8.014,149.488
C08676=1117.335,98.695,-57.357,-179.861,8.018,149.488
C08677=1117.330,98.944,-57.377,-179.859,8.022,149.488
C08678=1117.326,99.193,-57.396,-179.857,8.026,149.489
C08679=1117.321,99.443,-57.414,-179.855,8.030,149.489
C08680=1117.316,99.692,-57.433,-179.854,8.033,149.490
C08681=1117.311,99.941,-57.453,-179.852,8.037,149.490
C08682=1117.306,100.191,-57.471,-179.850,8.041,149.490
C08683=1117.302,100.440,-57.490,-179.849,8.045,149.491
C08684=1117.296,100.689,-57.510,-179.847,8.049,149.491
C08685=1117.292,100.938,-57.529,-179.844,8.053,149.491
C08686=1117.287,101.188,-57.547,-179.843,8.057,149.492
C08687=1117.282,101.437,-57.567,-179.841,8.061,149.492
C08688=1117.277,101.686,-57.586,-179.839,8.064,149.492
C08689=1117.272,101.935,-57.605,-179.837,8.068,149.493
C08690=1117.268,102.184,-57.624,-179.836,8.072,149.493
C08691=1117.263,102.433,-57.644,-179.834,8.075,149.494
C08692=1117.259,102.649,-57.660,-179.832,8.079,149.494
C08693=1117.255,102.865,-57.676,-179.831,8.082,149.494
C08694=1117.250,103.082,-57.694,-179.829,8.086,149.494
C08695=1117.246,103.297,-57.710,-179.828,8.089,149.495
C08696=1117.242,103.513,-57.726,-179.826,8.092,149.495
C08697=1117.238,103.730,-57.743,-179.824,8.096,149.495
C08698=1117.234,103.945,-57.759,-179.823,8.099,149.496
C08699=1117.229,104.162,-57.777,-179.821,8.102,149.496
C08700=1117.225,104.411,-57.795,-179.819,8.106,149.496
C08701=1117.220,104.660,-57.815,-179.817,8.110,149.497
C08702=1117.215,104.909,-57.834,-179.815,8.113,149.497
C08703=1117.211,105.158,-57.854,-179.813,8.118,149.497
C08704=1117.206,105.408,-57.873,-179.811,8.121,149.497
C08705=1117.200,105.657,-57.892,-179.809,8.125,149.498
C08706=1117.196,105.906,-57.912,-179.807,8.129,149.498
C08707=1117.191,106.155,-57.931,-179.805,8.133,149.499
C08708=1117.186,106.404,-57.950,-179.803,8.136,149.499
C08709=1117.182,106.654,-57.970,-179.801,8.140,149.499
C08710=1117.176,106.903,-57.989,-179.799,8.144,149.499
C08711=1117.172,107.152,-58.008,-179.797,8.148,149.500
C08712=1117.168,107.402,-58.028,-179.795,8.151,149.500
C08713=1117.162,107.651,-58.047,-179.793,8.156,149.500
C08714=1117.158,107.900,-58.068,-179.791,8.159,149.501
C08715=1117.152,108.148,-58.087,-179.788,8.163,149.501
C08716=1117.148,108.398,-58.106,-179.786,8.166,149.501
C08717=1117.144,108.647,-58.126,-179.784,8.170,149.501
C08718=1117.138,108.896,-58.145,-179.782,8.175,149.502
C08719=1117.134,109.146,-58.165,-179.780,8.178,149.502
C08720=1117.129,109.395,-58.185,-179.778,8.182,149.502
C08721=1117.124,109.644,-58.205,-179.776,8.185,149.502
C08722=1117.119,109.893,-58.224,-179.773,8.189,149.503
C08723=1117.114,110.143,-58.244,-179.771,8.193,149.503
C08724=1117.110,110.392,-58.263,-179.770,8.197,149.503
C08725=1117.105,110.640,-58.283,-179.767,8.201,149.503
C08726=1117.101,110.890,-58.302,-179.765,8.205,149.504
C08727=1117.096,111.139,-58.322,-179.763,8.208,149.504
C08728=1117.091,111.388,-58.342,-179.761,8.212,149.504
C08729=1117.086,111.637,-58.362,-179.759,8.215,149.504
C08730=1117.081,111.887,-58.381,-179.758,8.218,149.505
C08731=1117.077,112.136,-58.401,-179.756,8.222,149.505
C08732=1117.072,112.384,-58.421,-179.754,8.225,149.505
C08733=1117.067,112.634,-58.441,-179.752,8.229,149.506
C08734=1117.062,112.883,-58.461,-179.750,8.233,149.506
C08735=1117.058,113.133,-58.481,-179.748,8.235,149.506
C08736=1117.052,113.381,-58.500,-179.747,8.239,149.507
C08737=1117.048,113.630,-58.520,-179.745,8.243,149.507
C08738=1117.043,113.880,-58.540,-179.743,8.246,149.507
C08739=1117.038,114.130,-58.560,-179.741,8.250,149.507
C08740=1117.034,114.378,-58.580,-179.739,8.254,149.508
C08741=1117.029,114.627,-58.599,-179.738,8.256,149.508
C08742=1117.024,114.876,-58.620,-179.736,8.260,149.508
C08743=1117.019,115.126,-58.639,-179.733,8.263,149.508
C08744=1117.015,115.375,-58.660,-179.732,8.267,149.509
C08745=1117.010,115.624,-58.679,-179.730,8.271,149.509
C08746=1117.005,115.873,-58.699,-179.728,8.273,149.509
C08747=1117.000,116.122,-58.720,-179.727,8.277,149.510
C08748=1116.996,116.336,-58.737,-179.725,8.280,149.510
C08749=1116.992,116.550,-58.754,-179.723,8.283,149.510
C08750=1116.988,116.765,-58.771,-179.722,8.286,149.510
C08751=1116.984,116.979,-58.788,-179.720,8.289,149.511
C08752=1116.979,117.192,-58.806,-179.719,8.292,149.511
C08753=1116.976,117.407,-58.824,-179.717,8.295,149.511
C08754=1116.971,117.621,-58.840,-179.715,8.298,149.511
C08755=1116.967,117.835,-58.858,-179.714,8.301,149.511
C08756=1116.963,118.084,-58.878,-179.712,8.304,149.512
C08757=1116.958,118.334,-58.898,-179.710,8.308,149.512
C08758=1116.953,118.583,-58.918,-179.709,8.311,149.512
C08759=1116.949,118.832,-58.938,-179.707,8.314,149.513
C08760=1116.944,119.081,-58.958,-179.705,8.318,149.513
C08761=1116.939,119.329,-58.978,-179.703,8.322,149.513
C08762=1116.934,119.579,-58.999,-179.702,8.324,149.513
C08763=1116.929,119.828,-59.019,-179.700,8.328,149.514
C08764=1116.925,120.077,-59.039,-179.698,8.331,149.514
C08765=1116.920,120.326,-59.060,-179.697,8.334,149.514
C08766=1116.916,120.576,-59.079,-179.695,8.338,149.515
C08767=1116.910,120.825,-59.100,-179.692,8.341,149.515
C08768=1116.906,121.074,-59.120,-179.690,8.345,149.515
C08769=1116.901,121.323,-59.140,-179.689,8.348,149.515
C08770=1116.897,121.572,-59.161,-179.687,8.351,149.516
C08771=1116.892,121.822,-59.181,-179.685,8.355,149.516
C08772=1116.887,122.071,-59.202,-179.683,8.358,149.516
C08773=1116.882,122.319,-59.222,-179.682,8.361,149.516
C08774=1116.877,122.568,-59.242,-179.680,8.365,149.517
C08775=1116.872,122.818,-59.262,-179.678,8.369,149.517
C08776=1116.868,123.067,-59.283,-179.677,8.371,149.517
C08777=1116.863,123.316,-59.303,-179.675,8.375,149.517
C08778=1116.858,123.565,-59.324,-179.673,8.379,149.518
C08779=1116.854,123.814,-59.345,-179.671,8.382,149.518
C08780=1116.849,124.063,-59.364,-179.669,8.385,149.518
C08781=1116.844,124.313,-59.385,-179.667,8.388,149.519
C08782=1116.839,124.562,-59.406,-179.665,8.392,149.519
C08783=1116.835,124.811,-59.426,-179.664,8.395,149.519
C08784=1116.830,125.060,-59.447,-179.662,8.398,149.519
C08785=1116.825,125.309,-59.467,-179.660,8.402,149.520
C08786=1116.821,125.558,-59.488,-179.659,8.405,149.520
C08787=1116.816,125.807,-59.509,-179.657,8.408,149.520
C08788=1116.811,126.056,-59.529,-179.655,8.412,149.521
C08789=1116.807,126.305,-59.549,-179.654,8.415,149.521
C08790=1116.802,126.554,-59.570,-179.652,8.418,149.521
C08791=1116.797,126.803,-59.591,-179.650,8.422,149.521
C08792=1116.792,127.052,-59.612,-179.648,8.426,149.522
C08793=1116.788,127.302,-59.632,-179.646,8.428,149.522
C08794=1116.784,127.551,-59.653,-179.644,8.432,149.522
C08795=1116.779,127.800,-59.674,-179.643,8.436,149.523
C08796=1116.774,128.049,-59.694,-179.641,8.438,149.523
C08797=1116.769,128.298,-59.715,-179.639,8.442,149.523
C08798=1116.765,128.547,-59.735,-179.637,8.445,149.523
C08799=1116.759,128.797,-59.756,-179.636,8.448,149.524
C08800=1116.755,129.046,-59.777,-179.634,8.452,149.524
C08801=1116.750,129.295,-59.798,-179.632,8.455,149.524
C08802=1116.745,129.544,-59.818,-179.631,8.458,149.524
C08803=1116.740,129.793,-59.839,-179.629,8.462,149.525
C08804=1116.737,130.007,-59.858,-179.627,8.465,149.525
C08805=1116.733,130.221,-59.875,-179.626,8.467,149.525
C08806=1116.728,130.434,-59.892,-179.625,8.470,149.525
C08807=1116.725,130.649,-59.910,-179.623,8.473,149.526
C08808=1116.720,130.862,-59.929,-179.621,8.476,149.526
C08809=1116.716,131.077,-59.947,-179.620,8.479,149.526
C08810=1116.712,131.291,-59.964,-179.618,8.482,149.526
C08811=1116.709,131.505,-59.983,-179.617,8.485,149.527
C08812=1116.704,131.754,-60.004,-179.615,8.488,149.527
C08813=1116.699,132.003,-60.024,-179.614,8.491,149.527
C08814=1116.694,132.252,-60.045,-179.612,8.495,149.527
C08815=1116.689,132.501,-60.066,-179.610,8.498,149.528
C08816=1116.685,132.750,-60.087,-179.609,8.501,149.528
C08817=1116.680,133.000,-60.108,-179.606,8.505,149.528
C08818=1116.676,133.249,-60.129,-179.605,8.507,149.529
C08819=1116.671,133.497,-60.150,-179.603,8.511,149.529
C08820=1116.666,133.746,-60.171,-179.601,8.515,149.529
C08821=1116.661,133.995,-60.192,-179.600,8.517,149.529
C08822=1116.656,134.245,-60.213,-179.598,8.521,149.530
C08823=1116.652,134.494,-60.234,-179.596,8.525,149.530
C08824=1116.647,134.743,-60.255,-179.595,8.528,149.530
C08825=1116.642,134.992,-60.276,-179.593,8.531,149.531
C08826=1116.638,135.241,-60.297,-179.591,8.535,149.531
C08827=1116.633,135.490,-60.318,-179.590,8.538,149.531
C08828=1116.628,135.738,-60.340,-179.588,8.542,149.532
C08829=1116.624,135.988,-60.361,-179.586,8.544,149.532
C08830=1116.619,136.237,-60.381,-179.584,8.548,149.532
C08831=1116.614,136.486,-60.403,-179.583,8.552,149.533
C08832=1116.610,136.735,-60.424,-179.581,8.554,149.533
C08833=1116.605,136.984,-60.446,-179.579,8.558,149.533
C08834=1116.600,137.234,-60.467,-179.578,8.562,149.534
C08835=1116.595,137.483,-60.488,-179.576,8.564,149.534
C08836=1116.591,137.731,-60.509,-179.575,8.568,149.534
C08837=1116.586,137.980,-60.530,-179.572,8.572,149.534
C08838=1116.581,138.230,-60.552,-179.571,8.574,149.535
C08839=1116.577,138.479,-60.572,-179.569,8.578,149.535
C08840=1116.572,138.727,-60.594,-179.568,8.581,149.535
C08841=1116.568,138.977,-60.615,-179.566,8.585,149.536
C08842=1116.563,139.226,-60.637,-179.564,8.588,149.536
C08843=1116.558,139.475,-60.658,-179.563,8.591,149.536
C08844=1116.553,139.723,-60.679,-179.561,8.595,149.537
C08845=1116.549,139.973,-60.701,-179.559,8.598,149.537
C08846=1116.544,140.222,-60.722,-179.558,8.602,149.537
C08847=1116.539,140.471,-60.743,-179.556,8.605,149.538
C08848=1116.535,140.720,-60.764,-179.555,8.608,149.538
C08849=1116.530,140.969,-60.786,-179.553,8.612,149.538
C08850=1116.525,141.218,-60.808,-179.551,8.615,149.538
C08851=1116.520,141.467,-60.828,-179.550,8.618,149.539
C08852=1116.516,141.716,-60.851,-179.548,8.622,149.539
C08853=1116.511,141.965,-60.872,-179.547,8.625,149.540
C08854=1116.507,142.214,-60.893,-179.545,8.628,149.540
C08855=1116.502,142.463,-60.915,-179.543,8.632,149.540
C08856=1116.498,142.712,-60.936,-179.542,8.635,149.540
C08857=1116.492,142.961,-60.957,-179.540,8.639,149.541
C08858=1116.488,143.210,-60.979,-179.538,8.642,149.541
C08859=1116.483,143.459,-61.001,-179.537,8.645,149.542
C08860=1116.480,143.674,-61.019,-179.535,8.648,149.542
C08861=1116.475,143.887,-61.038,-179.534,8.651,149.542
C08862=1116.472,144.101,-61.056,-179.532,8.655,149.542
C08863=1116.468,144.315,-61.075,-179.531,8.657,149.543
C08864=1116.464,144.528,-61.093,-179.529,8.660,149.543
C08865=1116.459,144.743,-61.112,-179.528,8.663,149.543
C08866=1116.456,144.957,-61.130,-179.527,8.666,149.544
C08867=1116.451,145.170,-61.149,-179.526,8.669,149.544
C08868=1116.447,145.420,-61.171,-179.524,8.672,149.544
C08869=1116.442,145.668,-61.193,-179.521,8.677,149.544
C08870=1116.437,145.917,-61.214,-179.519,8.680,149.545
C08871=1116.433,146.167,-61.236,-179.517,8.684,149.545
C08872=1116.428,146.416,-61.257,-179.514,8.688,149.545
C08873=1116.423,146.665,-61.279,-179.512,8.691,149.545
C08874=1116.419,146.914,-61.301,-179.510,8.695,149.546
C08875=1116.414,147.162,-61.323,-179.508,8.698,149.546
C08876=1116.409,147.412,-61.345,-179.505,8.703,149.546
C08877=1116.405,147.660,-61.366,-179.503,8.706,149.546
C08878=1116.400,147.910,-61.388,-179.501,8.710,149.547
C08879=1116.395,148.158,-61.410,-179.499,8.713,149.547
C08880=1116.391,148.408,-61.431,-179.496,8.717,149.547
C08881=1116.386,148.657,-61.453,-179.494,8.721,149.547
C08882=1116.382,148.906,-61.475,-179.492,8.724,149.548
C08883=1116.377,149.155,-61.497,-179.490,8.728,149.548
C08884=1116.372,149.403,-61.519,-179.488,8.731,149.548
C08885=1116.368,149.653,-61.541,-179.485,8.735,149.548
C08886=1116.362,149.902,-61.563,-179.483,8.739,149.548
C08887=1116.358,150.151,-61.585,-179.481,8.742,149.548
C08888=1116.353,150.399,-61.607,-179.479,8.746,149.549
C08889=1116.349,150.648,-61.629,-179.477,8.749,149.549
C08890=1116.344,150.897,-61.651,-179.474,8.753,149.549
C08891=1116.340,151.146,-61.673,-179.472,8.756,149.549
C08892=1116.335,151.395,-61.695,-179.469,8.760,149.549
C08893=1116.330,151.645,-61.717,-179.467,8.764,149.550
C08894=1116.325,151.893,-61.739,-179.465,8.767,149.550
C08895=1116.321,152.143,-61.761,-179.463,8.770,149.550
C08896=1116.316,152.391,-61.783,-179.461,8.774,149.550
C08897=1116.312,152.640,-61.806,-179.458,8.777,149.550
C08898=1116.307,152.890,-61.828,-179.456,8.781,149.551
C08899=1116.302,153.138,-61.850,-179.454,8.784,149.551
C08900=1116.298,153.388,-61.872,-179.452,8.787,149.551
C08901=1116.293,153.636,-61.894,-179.449,8.791,149.551
C08902=1116.288,153.885,-61.917,-179.447,8.795,149.551
C08903=1116.283,154.134,-61.939,-179.444,8.798,149.551
C08904=1116.279,154.383,-61.961,-179.442,8.802,149.552
C08905=1116.274,154.632,-61.982,-179.440,8.805,149.552
C08906=1116.270,154.881,-62.006,-179.438,8.808,149.552
C08907=1116.265,155.130,-62.028,-179.436,8.812,149.552
C08908=1116.260,155.379,-62.050,-179.434,8.815,149.552
C08909=1116.256,155.628,-62.073,-179.431,8.818,149.552
C08910=1116.251,155.877,-62.095,-179.429,8.822,149.553
C08911=1116.247,156.126,-62.117,-179.427,8.825,149.553
C08912=1116.243,156.375,-62.139,-179.424,8.828,149.553
C08913=1116.237,156.624,-62.162,-179.422,8.832,149.553
C08914=1116.233,156.873,-62.184,-179.420,8.835,149.553
C08915=1116.229,157.122,-62.206,-179.418,8.838,149.553
C08916=1116.224,157.335,-62.225,-179.416,8.841,149.554
C08917=1116.220,157.549,-62.245,-179.414,8.844,149.554
C08918=1116.216,157.763,-62.264,-179.412,8.847,149.554
C08919=1116.213,157.977,-62.284,-179.410,8.850,149.554
C08920=1116.208,158.191,-62.303,-179.408,8.852,149.554
C08921=1116.204,158.405,-62.322,-179.406,8.855,149.554
C08922=1116.201,158.618,-62.342,-179.404,8.858,149.554
C08923=1116.196,158.833,-62.361,-179.402,8.861,149.555
C08924=1116.192,159.081,-62.383,-179.400,8.864,149.555
C08925=1116.187,159.330,-62.406,-179.398,8.867,149.555
C08926=1116.183,159.579,-62.429,-179.395,8.871,149.555
C08927=1116.178,159.828,-62.450,-179.393,8.874,149.555
C08928=1116.173,160.077,-62.474,-179.391,8.877,149.555
C08929=1116.169,160.325,-62.497,-179.389,8.881,149.555
C08930=1116.164,160.574,-62.519,-179.386,8.884,149.555
C08931=1116.160,160.823,-62.542,-179.385,8.886,149.556
C08932=1116.155,161.073,-62.564,-179.382,8.890,149.556
C08933=1116.151,161.321,-62.587,-179.380,8.893,149.556
C08934=1116.145,161.570,-62.609,-179.377,8.896,149.556
C08935=1116.141,161.819,-62.632,-179.375,8.899,149.556
C08936=1116.137,162.068,-62.655,-179.373,8.903,149.556
C08937=1116.132,162.318,-62.677,-179.370,8.906,149.556
C08938=1116.127,162.566,-62.700,-179.368,8.909,149.556
C08939=1116.123,162.815,-62.723,-179.366,8.912,149.556
C08940=1116.118,163.064,-62.746,-179.364,8.915,149.557
C08941=1116.114,163.313,-62.769,-179.362,8.918,149.557
C08942=1116.109,163.561,-62.792,-179.359,8.921,149.557
C08943=1116.104,163.810,-62.815,-179.357,8.925,149.557
C08944=1116.100,164.060,-62.837,-179.355,8.928,149.557
C08945=1116.095,164.309,-62.860,-179.353,8.931,149.557
C08946=1116.091,164.557,-62.883,-179.351,8.934,149.557
C08947=1116.086,164.806,-62.906,-179.348,8.937,149.557
C08948=1116.082,165.054,-62.929,-179.346,8.940,149.558
C08949=1116.077,165.304,-62.952,-179.344,8.944,149.558
C08950=1116.072,165.553,-62.975,-179.341,8.947,149.558
C08951=1116.068,165.802,-62.998,-179.340,8.949,149.558
C08952=1116.064,166.051,-63.021,-179.337,8.952,149.558
C08953=1116.058,166.299,-63.044,-179.335,8.956,149.558
C08954=1116.054,166.549,-63.066,-179.332,8.959,149.558
C08955=1116.049,166.798,-63.089,-179.330,8.962,149.558
C08956=1116.045,167.047,-63.113,-179.328,8.965,149.559
C08957=1116.041,167.295,-63.136,-179.326,8.968,149.559
C08958=1116.036,167.544,-63.159,-179.323,8.971,149.559
C08959=1116.031,167.793,-63.182,-179.321,8.975,149.559
C08960=1116.026,168.042,-63.205,-179.319,8.978,149.559
C08961=1116.022,168.290,-63.228,-179.317,8.980,149.559
C08962=1116.017,168.540,-63.251,-179.315,8.983,149.559
C08963=1116.013,168.789,-63.275,-179.312,8.987,149.559
C08964=1116.009,169.037,-63.297,-179.310,8.990,149.559
C08965=1116.004,169.286,-63.321,-179.308,8.992,149.559
C08966=1115.999,169.535,-63.344,-179.306,8.996,149.559
C08967=1115.994,169.784,-63.367,-179.303,8.999,149.560
C08968=1115.989,170.033,-63.391,-179.301,9.002,149.560
C08969=1115.985,170.281,-63.413,-179.299,9.004,149.560
C08970=1115.981,170.530,-63.437,-179.297,9.008,149.560
C08971=1115.976,170.779,-63.460,-179.295,9.011,149.560
C08972=1115.972,170.993,-63.480,-179.293,9.013,149.560
C08973=1115.968,171.207,-63.500,-179.291,9.016,149.560
C08974=1115.964,171.420,-63.520,-179.289,9.018,149.560
C08975=1115.960,171.634,-63.540,-179.288,9.021,149.560
C08976=1115.957,171.848,-63.560,-179.285,9.024,149.560
C08977=1115.952,172.062,-63.580,-179.283,9.026,149.560
C08978=1115.949,172.276,-63.600,-179.281,9.028,149.560
C08979=1115.945,172.489,-63.620,-179.280,9.031,149.561
C08980=1115.940,172.738,-63.643,-179.277,9.034,149.561
C08981=1115.936,172.987,-63.667,-179.275,9.037,149.561
C08982=1115.931,173.236,-63.691,-179.273,9.040,149.561
C08983=1115.926,173.485,-63.714,-179.271,9.043,149.561
C08984=1115.922,173.734,-63.738,-179.268,9.046,149.561
C08985=1115.918,173.983,-63.760,-179.267,9.049,149.561
C08986=1115.913,174.231,-63.784,-179.264,9.052,149.561
C08987=1115.909,174.480,-63.808,-179.262,9.055,149.561
C08988=1115.904,174.729,-63.831,-179.260,9.058,149.561
C08989=1115.899,174.978,-63.854,-179.258,9.061,149.562
C08990=1115.895,175.226,-63.879,-179.255,9.064,149.562
C08991=1115.890,175.476,-63.902,-179.253,9.067,149.562
C08992=1115.885,175.725,-63.925,-179.251,9.070,149.562
C08993=1115.881,175.973,-63.949,-179.249,9.073,149.562
C08994=1115.876,176.222,-63.973,-179.247,9.075,149.562
C08995=1115.872,176.471,-63.996,-179.245,9.079,149.562
C08996=1115.867,176.719,-64.020,-179.242,9.082,149.562
C08997=1115.862,176.968,-64.043,-179.240,9.084,149.562
C08998=1115.858,177.218,-64.067,-179.238,9.088,149.563
C08999=1115.853,177.466,-64.091,-179.236,9.091,149.563
C09000=1115.849,177.715,-64.114,-179.234,9.093,149.563
C09001=1115.844,177.963,-64.138,-179.232,9.097,149.563
C09002=1115.840,178.212,-64.162,-179.230,9.099,149.563
C09003=1115.835,178.461,-64.185,-179.227,9.102,149.563
C09004=1115.830,178.710,-64.209,-179.225,9.106,149.563
C09005=1115.826,178.959,-64.232,-179.223,9.108,149.563
C09006=1115.822,179.208,-64.257,-179.221,9.111,149.563
C09007=1115.817,179.457,-64.280,-179.219,9.115,149.564
C09008=1115.813,179.705,-64.304,-179.216,9.118,149.564
C09009=1115.808,179.954,-64.328,-179.214,9.121,149.564
C09010=1115.804,180.203,-64.352,-179.211,9.124,149.564
C09011=1115.799,180.452,-64.375,-179.208,9.127,149.564
C09012=1115.795,180.700,-64.399,-179.206,9.130,149.564
C09013=1115.789,180.950,-64.423,-179.203,9.133,149.564
C09014=1115.785,181.199,-64.448,-179.201,9.136,149.564
C09015=1115.781,181.447,-64.472,-179.198,9.139,149.564
C09016=1115.776,181.696,-64.495,-179.196,9.142,149.564
C09017=1115.772,181.945,-64.519,-179.193,9.145,149.564
C09018=1115.767,182.194,-64.542,-179.191,9.148,149.564
C09019=1115.763,182.442,-64.567,-179.188,9.152,149.564
C09020=1115.758,182.692,-64.592,-179.185,9.155,149.564
C09021=1115.754,182.941,-64.615,-179.183,9.158,149.564
C09022=1115.749,183.189,-64.639,-179.180,9.161,149.564
C09023=1115.745,183.437,-64.663,-179.178,9.164,149.564
C09024=1115.740,183.686,-64.686,-179.175,9.167,149.564
C09025=1115.735,183.935,-64.711,-179.173,9.169,149.564
C09026=1115.731,184.184,-64.736,-179.171,9.173,149.564
C09027=1115.727,184.433,-64.760,-179.168,9.176,149.564
C09028=1115.722,184.647,-64.780,-179.167,9.178,149.564
C09029=1115.719,184.859,-64.801,-179.164,9.181,149.564
C09030=1115.715,185.074,-64.821,-179.162,9.183,149.564
C09031=1115.711,185.287,-64.842,-179.160,9.185,149.564
C09032=1115.707,185.500,-64.863,-179.158,9.188,149.564
C09033=1115.703,185.715,-64.884,-179.155,9.191,149.564
C09034=1115.700,185.928,-64.904,-179.153,9.193,149.564
C09035=1115.696,186.141,-64.925,-179.152,9.195,149.564
C09036=1115.691,186.390,-64.949,-179.149,9.199,149.564
C09037=1115.686,186.639,-64.974,-179.147,9.201,149.564
C09038=1115.682,186.888,-64.998,-179.145,9.204,149.565
C09039=1115.678,187.136,-65.022,-179.142,9.207,149.565
C09040=1115.673,187.385,-65.047,-179.140,9.209,149.565
C09041=1115.669,187.634,-65.071,-179.138,9.213,149.565
C09042=1115.664,187.883,-65.095,-179.135,9.216,149.565
C09043=1115.659,188.131,-65.120,-179.133,9.218,149.565
C09044=1115.654,188.380,-65.143,-179.131,9.221,149.565
C09045=1115.650,188.630,-65.168,-179.128,9.224,149.565
C09046=1115.646,188.878,-65.192,-179.126,9.227,149.565
C09047=1115.641,189.127,-65.216,-179.124,9.230,149.565
C09048=1115.637,189.376,-65.241,-179.122,9.232,149.565
C09049=1115.632,189.624,-65.265,-179.119,9.235,149.565
C09050=1115.627,189.873,-65.290,-179.117,9.238,149.565
C09051=1115.623,190.122,-65.314,-179.115,9.241,149.565
C09052=1115.619,190.371,-65.339,-179.112,9.244,149.565
C09053=1115.614,190.619,-65.363,-179.111,9.246,149.565
C09054=1115.610,190.868,-65.388,-179.108,9.249,149.565
C09055=1115.605,191.117,-65.412,-179.106,9.251,149.565
C09056=1115.600,191.366,-65.436,-179.104,9.255,149.565
C09057=1115.596,191.614,-65.462,-179.102,9.257,149.565
C09058=1115.592,191.863,-65.486,-179.099,9.260,149.565
C09059=1115.587,192.112,-65.511,-179.098,9.263,149.566
C09060=1115.583,192.361,-65.535,-179.095,9.266,149.566
C09061=1115.578,192.609,-65.560,-179.093,9.268,149.566
C09062=1115.573,192.858,-65.584,-179.091,9.270,149.566
C09063=1115.569,193.107,-65.609,-179.089,9.274,149.566
C09064=1115.564,193.356,-65.633,-179.087,9.276,149.566
C09065=1115.560,193.604,-65.659,-179.085,9.279,149.566
C09066=1115.556,193.853,-65.683,-179.083,9.282,149.566
C09067=1115.551,194.102,-65.708,-179.081,9.285,149.566
C09068=1115.547,194.351,-65.732,-179.079,9.287,149.566
C09069=1115.542,194.599,-65.757,-179.077,9.290,149.566
C09070=1115.537,194.847,-65.782,-179.075,9.293,149.567
C09071=1115.533,195.097,-65.807,-179.073,9.295,149.567
C09072=1115.528,195.345,-65.831,-179.071,9.298,149.567
C09073=1115.524,195.594,-65.856,-179.069,9.301,149.567
C09074=1115.519,195.843,-65.881,-179.067,9.304,149.567
C09075=1115.516,196.092,-65.906,-179.065,9.307,149.567
C09076=1115.511,196.340,-65.930,-179.063,9.309,149.567
C09077=1115.505,196.589,-65.955,-179.060,9.312,149.567
C09078=1115.502,196.838,-65.980,-179.057,9.316,149.567
C09079=1115.497,197.086,-66.005,-179.055,9.319,149.567
C09080=1115.493,197.335,-66.029,-179.052,9.322,149.567
C09081=1115.488,197.584,-66.055,-179.049,9.326,149.567
C09082=1115.484,197.833,-66.080,-179.046,9.329,149.567
C09083=1115.480,198.081,-66.104,-179.043,9.332,149.567
C09084=1115.476,198.295,-66.126,-179.041,9.335,149.567
C09085=1115.472,198.508,-66.147,-179.038,9.338,149.567
C09086=1115.468,198.722,-66.168,-179.036,9.340,149.567
C09087=1115.464,198.935,-66.190,-179.033,9.343,149.567
C09088=1115.461,199.148,-66.212,-179.030,9.346,149.567
C09089=1115.456,199.362,-66.233,-179.027,9.349,149.567
C09090=1115.453,199.576,-66.254,-179.025,9.351,149.567
C09091=1115.449,199.789,-66.275,-179.022,9.354,149.567
C09092=1115.444,200.038,-66.301,-179.020,9.357,149.567
C09093=1115.439,200.286,-66.326,-179.017,9.360,149.567
C09094=1115.435,200.535,-66.352,-179.014,9.363,149.567
C09095=1115.431,200.784,-66.376,-179.011,9.366,149.567
C09096=1115.426,201.032,-66.401,-179.008,9.369,149.566
C09097=1115.422,201.281,-66.427,-179.005,9.372,149.566
C09098=1115.417,201.530,-66.452,-179.002,9.375,149.566
C09099=1115.413,201.779,-66.478,-178.999,9.377,149.566
C09100=1115.408,202.027,-66.502,-178.996,9.381,149.566
C09101=1115.404,202.276,-66.527,-178.993,9.384,149.566
C09102=1115.399,202.524,-66.553,-178.990,9.387,149.566
C09103=1115.395,202.774,-66.578,-178.987,9.390,149.566
C09104=1115.391,203.022,-66.604,-178.985,9.393,149.566
C09105=1115.387,203.270,-66.628,-178.982,9.395,149.566
C09106=1115.382,203.520,-66.653,-178.979,9.398,149.566
C09107=1115.377,203.768,-66.679,-178.976,9.401,149.565
C09108=1115.373,204.017,-66.705,-178.974,9.404,149.565
C09109=1115.368,204.266,-66.730,-178.970,9.408,149.565
C09110=1115.364,204.514,-66.755,-178.967,9.410,149.565
C09111=1115.359,204.763,-66.781,-178.964,9.413,149.565
C09112=1115.355,205.011,-66.806,-178.962,9.416,149.565
C09113=1115.350,205.260,-66.832,-178.959,9.419,149.565
C09114=1115.346,205.509,-66.857,-178.956,9.422,149.565
C09115=1115.341,205.757,-66.882,-178.953,9.424,149.565
C09116=1115.337,206.006,-66.908,-178.950,9.427,149.565
C09117=1115.332,206.255,-66.934,-178.947,9.430,149.565
C09118=1115.328,206.503,-66.959,-178.944,9.433,149.564
C09119=1115.323,206.752,-66.985,-178.942,9.436,149.565
